		IF ABS(axis.NcToPlc.ActTorque) > ABS(TorqueLimit) THEN
			//fbDetectTime(IN := TRUE,PT := DetectionTorqueTime); 
			fbDetectTime.IN := TRUE;
			IF fbDetectTime.Q THEN
				jog.JogForward := FALSE;
				jog.JogBackwards := FALSE;
				nState := nState + 1;
			END_IF
		ELSIF NOT jogOut.Busy AND jogOut.Error THEN
			Error := jogOut.Error;
			ErrorID := jogOut.ErrorID;
			jog.JogForward := FALSE;
			jog.JogBackwards := FALSE;
			nState := 0;
		ELSIF jogOut.CommandAborted THEN
			jog.JogForward := FALSE;
			jog.JogBackwards := FALSE;
		ELSE
			fbDetectTime.IN := FALSE;
			//fbDetectTime(IN := FALSE,PT := DetectionTorqueTime);
		END_IF
		
	2: // Stop motor
		stop.Execute := TRUE;
		
		IF stopOut.Busy AND stopOut.Done THEN
			stop.Execute := FALSE;
			Busy := FALSE;
			Done := TRUE;
			nState := 0;
			
		ELSIF NOT stopOut.Busy AND stopOut.Error THEN
			Error := stopOut.Error;
			ErrorId := stopOut.ErrorID;
			stop.Execute := FALSE;
			nState := 0;
		END_IF
END_CASE

IF axis.Status.Error THEN
	nState := 0;
END_IF

ACTION actMove:
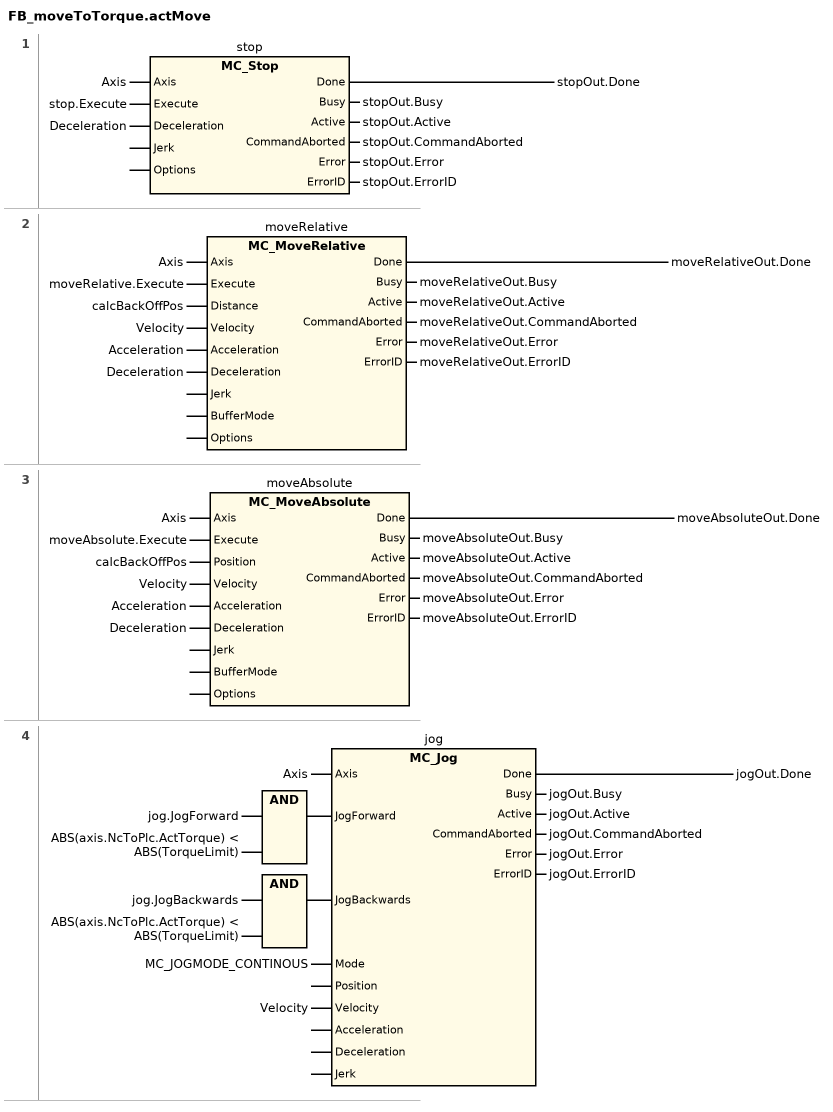
// NETWORK 1
stop(
    Axis := Axis,
    Execute := stop.Execute,
    Deceleration := Deceleration,
    Busy => stopOut.Busy,
    Active => stopOut.Active,
    CommandAborted => stopOut.CommandAborted,
    Error => stopOut.Error,
    ErrorID => stopOut.ErrorID); // MC_Stop
stopOut.Done := stop.Done;

// NETWORK 2
moveRelative(
    Axis := Axis,
    Execute := moveRelative.Execute,
    Distance := calcBackOffPos,
    Velocity := Velocity,
    Acceleration := Acceleration,
    Deceleration := Deceleration,
    Busy => moveRelativeOut.Busy,
    Active => moveRelativeOut.Active,
    CommandAborted => moveRelativeOut.CommandAborted,
    Error => moveRelativeOut.Error,
    ErrorID => moveRelativeOut.ErrorID); // MC_MoveRelative
moveRelativeOut.Done := moveRelative.Done;

// NETWORK 3
moveAbsolute(
    Axis := Axis,
    Execute := moveAbsolute.Execute,
    Position := calcBackOffPos,
    Velocity := Velocity,
    Acceleration := Acceleration,
    Deceleration := Deceleration,
    Busy => moveAbsoluteOut.Busy,
    Active => moveAbsoluteOut.Active,
    CommandAborted => moveAbsoluteOut.CommandAborted,
    Error => moveAbsoluteOut.Error,
    ErrorID => moveAbsoluteOut.ErrorID); // MC_MoveAbsolute
moveAbsoluteOut.Done := moveAbsolute.Done;

// NETWORK 4
jog(
    Axis := Axis,
    JogForward := jog.JogForward AND (ABS(axis.NcToPlc.ActTorque) < ABS(TorqueLimit)),
    JogBackwards := jog.JogBackwards AND (ABS(axis.NcToPlc.ActTorque) < ABS(TorqueLimit)),
    Mode := MC_JOGMODE_CONTINOUS,
    Velocity := Velocity,
    Busy => jogOut.Busy,
    Active => jogOut.Active,
    CommandAborted => jogOut.CommandAborted,
    Error => jogOut.Error,
    ErrorID => jogOut.ErrorID); // MC_Jog
jogOut.Done := jog.Done;
END_ACTION

END_FUNCTION_BLOCK

// ---- POUs/FUNCTIONS/FB_homeToTorque.TcPOU
FUNCTION_BLOCK FB_homeToTorque
VAR_IN_OUT
	Axis : AXIS_REF;					
END_VAR
VAR_INPUT
	Execute 		: BOOL;
	Direction 		: INT; // 0- PositiveDirection, 1- NegativeDirection
	Velocity 		: LREAL;
	Acceleration 	: LREAL;
	Deceleration 	: LREAL;
	SetPosition 	: LREAL;
	TimeLimit 		: TIME;
	TorqueLimit 	: LREAL;
	BackOffPos 		: LREAL;
END_VAR
VAR_OUTPUT
	Done 			: BOOL;
	Busy 			: BOOL;
	Active 			: BOOL;
	CommandAborted 	: BOOL;
	Error 			: BOOL;
	ErrorID 		: UDINT;
END_VAR
VAR
	nState 			: INT;
	fbExecute 		: R_TRIG;
	fbTimeout 		: TON;
	fbDetectTime 	: TON;
	
	readParameter 		: MC_ReadParameter;
	readParameterOut 	: ST_mcOutputs;
	
	writeParameter		: MC_WriteParameter;
	writeParameterOut 	: ST_mcOutputs;
	readValue 			: LREAL;
	
	parameter 	: MC_AxisParameter;	
	writeValue 	: LREAL;
	
	moveToTorque	: MC_TorqueControl;
	torqueOptions 	: ST_TorqueControlOptions;
	moveToTorqueOut : ST_mcOutputs;
	
	moveAbsolute	: MC_MoveAbsolute;
	moveAbsoluteOut : ST_mcOutputs;
	calcBackOffPos 	: LREAL;
	
	home	: MC_Home;
	homeOut : ST_mcOutputs;
	
	stop		: MC_Stop;
	stopOut 	: ST_mcOutputs;
	fPosition	: LREAL;

	jog		: MC_Jog;
	jogOut 	: ST_mcOutputs;
	
	moveRelative	: MC_MoveRelative;
	moveRelativeOut	: ST_mcOutputs;
END_VAR

fbExecute(CLK := Execute);
fbTimeout();
actHome();
actMode();
actMove();


CASE nState OF 
	0: //init
		IF NOT Execute THEN
		(* reset at falling edge of Execute *)
			Busy 					:= FALSE;
			Done					:= FALSE;
			CommandAborted 			:= FALSE;
			Error 					:= FALSE;
			ErrorID 				:= 0;
			fbTimeout.IN 			:= FALSE;
			readParameter.Enable 	:= FALSE;
			writeParameter.Execute	:= FALSE;
			stop.Execute		 	:= FALSE;
			home.Execute 			:= FALSE;
			moveAbsolute.Execute 	:= FALSE;
			jog.JogForward 			:= FALSE;
			jog.JogBackwards 		:= FALSE;
		END_IF
	
		IF fbExecute.Q THEN
			Busy := TRUE;
			nState := nState + 1;
		END_IF
		
	1:// Read soft limit switch to set back to when done
		CASE Direction OF 
			0: //mcPositiveDirection
		      	parameter := AxisMaxSoftPosLimit;
			1: //mcNegativeDirection
				parameter := AxisMinSoftPosLimit;
		END_CASE
		
		readParameter.Enable := TRUE;
		
		IF NOT readParameterOut.Busy AND readParameterOut.Done THEN
			readParameter.Enable := FALSE;
			nState := nState + 1;
		ELSIF NOT readParameterOut.Busy AND readParameterOut.Error THEN
			Error := readParameterOut.Error;
			ErrorId := readParameterOut.ErrorID;
			readParameter.Enable := FALSE;
			nState := 0;
		END_IF
		
	2: // Set soft limit switch to appropriate allowance
		CASE Direction OF
			0 : //mcPositiveDirection
				writeValue := 99999;
			1 : //mcNegativeDirection
				writeValue := -99999;
		END_CASE
		
		writeParameter.Execute := TRUE;
		
		IF NOT writeParameterOut.Busy AND writeParameterOut.Done THEN
			writeParameter.Execute := FALSE;
			nState := nState + 1;
		ELSIF NOT writeParameterOut.Busy AND writeParameterOut.Error THEN
			Error := writeParameterOut.Error;
			ErrorID := writeParameterOut.ErrorID;
			writeParameter.Execute := FALSE;
			nState := 0;
		END_IF
		
	3: //Execute MoveTowards Torque
		fbTimeout(IN:= TRUE, PT:= TimeLimit);
		
		CASE Direction OF
			0: //mcPositiveDirection 
				jog.JogForward := TRUE;
				jog.JogBackwards := FALSE;
			1: //mcNegativeDirection 
				jog.JogForward := FALSE;
				jog.JogBackwards := TRUE;
		END_CASE
			
		IF ABS(axis.NcToPlc.ActTorque) > ABS(TorqueLimit) THEN
			jog.JogForward := FALSE;
			jog.JogBackwards := FALSE;
			nState := nState + 1;
		ELSIF NOT jogOut.Busy AND jogOut.Error THEN
			Error := jogOut.Error;
			ErrorID := jogOut.ErrorID;
			jog.JogForward := FALSE;
			jog.JogBackwards := FALSE;
			nState := 0;
		END_IF
		
		// Timeout Error
		IF fbTimeout.Q THEN
			jog.JogForward := FALSE;
			jog.JogBackwards := FALSE;
			Error := TRUE;
			ErrorID := 1;
			nState := 0;
		END_IF
		
		CommandAborted := jogOut.CommandAborted;
	4://Stop motor 
		stop.Execute := TRUE;
		
		IF stopOut.Busy AND stopOut.Done THEN
			stop.Execute := FALSE;
			CASE Direction OF
				0: //mcPositiveDirection 
					calcBackOffPos := -BackOffPos;
				1: //mcNegativeDirection 
					calcBackOffPos := BackOffPos;
			END_CASE
			nState := nState + 1;
			
		ELSIF NOT stopOut.Busy AND stopOut.Error THEN
			Error := stopOut.Error;
			ErrorId := stopOut.ErrorID;
			stop.Execute := FALSE;
			nState := 0;
		END_IF
		
		CommandAborted := stopOut.CommandAborted;
	6: //Set homing state and counts
		IF axis.status.StandStill THEN
			home.Execute := TRUE;
		END_IF
		
		IF NOT homeOut.Busy AND homeOut.Done THEN
			home.Execute := FALSE;
			nState := nState + 1;
		ELSIF NOT homeOut.Busy AND homeOut.Error THEN
			Error := homeOut.Error;
			ErrorId := homeOut.ErrorID;
			home.Execute := FALSE;
			nState := 0;
		END_IF
		
		CommandAborted := homeOut.CommandAborted;
	5: //Move off home slightly
		IF axis.status.StandStill THEN
			moveRelative.Execute := TRUE;
		END_IF
		
		IF NOT moveRelativeOut.Busy AND moveRelativeOut.Done THEN
			moveRelative.Execute := FALSE;
			nState := nState + 1;
		ELSIF NOT moveRelativeOut.Busy AND moveRelativeOut.Error THEN
			Error := moveRelativeOut.Error;
			ErrorId := moveRelativeOut.ErrorID;
			moveRelative.Execute := FALSE;
			nState := 0;
		END_IF
		
		CommandAborted := moveRelativeOut.CommandAborted;
	7: // Write limit switch to original Value
		writeValue := SetPosition;
		writeParameter.Execute := TRUE;
		
		IF NOT writeParameterOut.Busy AND writeParameterOut.Done THEN
			writeParameter.Execute := FALSE;
			Busy := FALSE;
			Done := TRUE;
			nState := 0;
		ELSIF NOT writeParameterOut.Busy AND writeParameterOut.Error THEN
			Error := writeParameterOut.Error;
			ErrorID := writeParameterOut.ErrorID;
			writeParameter.Execute := FALSE;
			nState := 0;
		END_IF
END_CASE

IF axis.Status.Error THEN
	nState := 0;
END_IF

ACTION actHome:
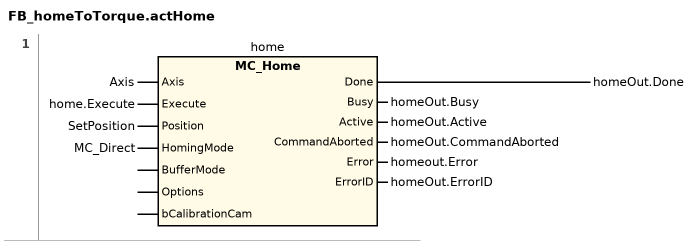
// NETWORK 1
home(
    Axis := Axis,
    Execute := home.Execute,
    Position := SetPosition,
    HomingMode := MC_Direct,
    Busy => homeOut.Busy,
    Active => homeOut.Active,
    CommandAborted => homeOut.CommandAborted,
    Error => homeout.Error,
    ErrorID => homeOut.ErrorID); // MC_Home
homeOut.Done := home.Done;
END_ACTION

ACTION actMode:
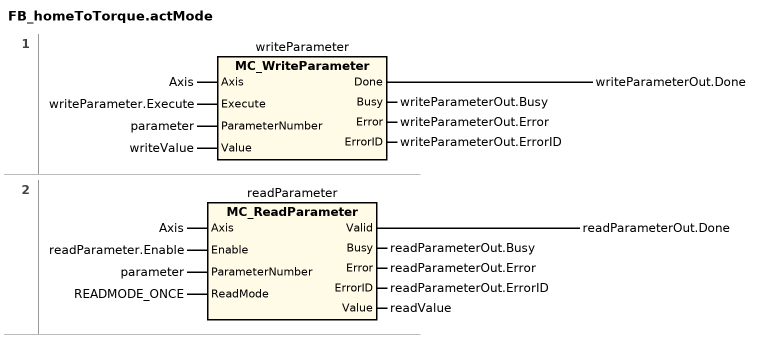
// NETWORK 1
writeParameter(
    Axis := Axis,
    Execute := writeParameter.Execute,
    ParameterNumber := parameter,
    Value := writeValue,
    Busy => writeParameterOut.Busy,
    Error => writeParameterOut.Error,
    ErrorID => writeParameterOut.ErrorID); // MC_WriteParameter
writeParameterOut.Done := writeParameter.Done;

// NETWORK 2
readParameter(
    Axis := Axis,
    Enable := readParameter.Enable,
    ParameterNumber := parameter,
    ReadMode := READMODE_ONCE,
    Busy => readParameterOut.Busy,
    Error => readParameterOut.Error,
    ErrorID => readParameterOut.ErrorID,
    Value => readValue); // MC_ReadParameter
readParameterOut.Done := readParameter.Valid;
END_ACTION

ACTION actMove:
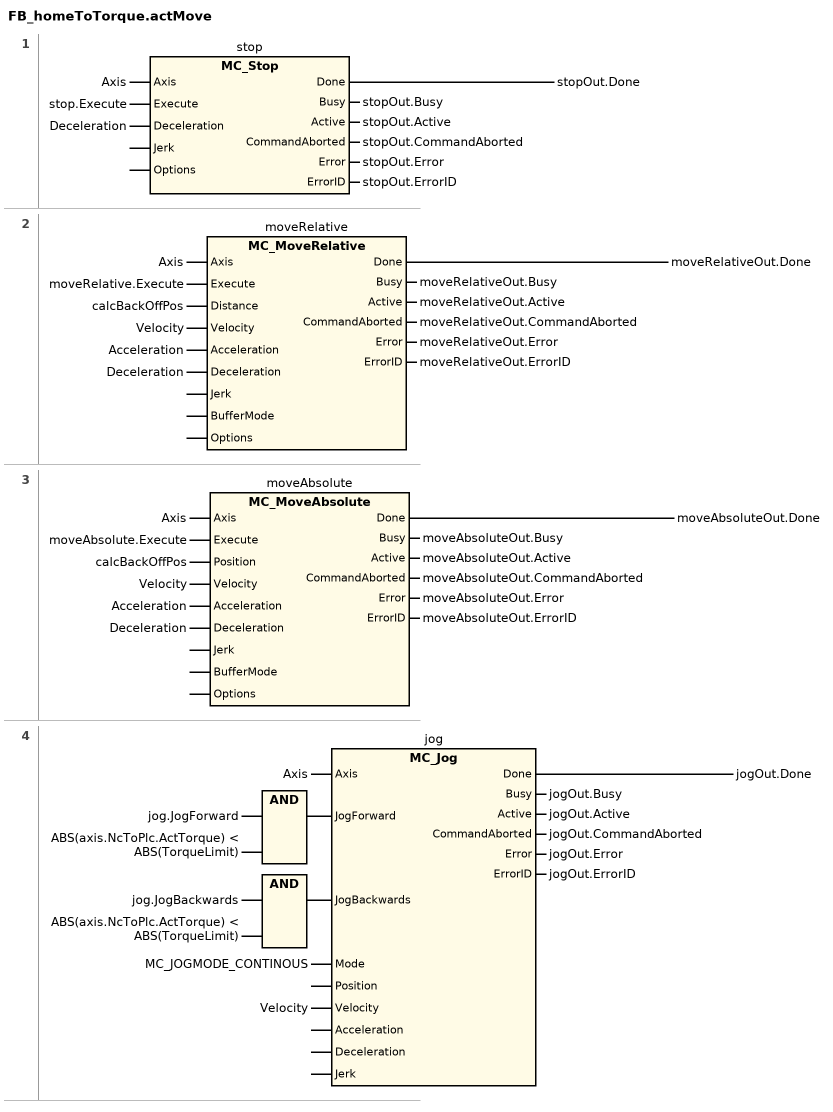
// NETWORK 1
stop(
    Axis := Axis,
    Execute := stop.Execute,
    Deceleration := Deceleration,
    Busy => stopOut.Busy,
    Active => stopOut.Active,
    CommandAborted => stopOut.CommandAborted,
    Error => stopOut.Error,
    ErrorID => stopOut.ErrorID); // MC_Stop
stopOut.Done := stop.Done;

// NETWORK 2
moveRelative(
    Axis := Axis,
    Execute := moveRelative.Execute,
    Distance := calcBackOffPos,
    Velocity := Velocity,
    Acceleration := Acceleration,
    Deceleration := Deceleration,
    Busy => moveRelativeOut.Busy,
    Active => moveRelativeOut.Active,
    CommandAborted => moveRelativeOut.CommandAborted,
    Error => moveRelativeOut.Error,
    ErrorID => moveRelativeOut.ErrorID); // MC_MoveRelative
moveRelativeOut.Done := moveRelative.Done;

// NETWORK 3
moveAbsolute(
    Axis := Axis,
    Execute := moveAbsolute.Execute,
    Position := calcBackOffPos,
    Velocity := Velocity,
    Acceleration := Acceleration,
    Deceleration := Deceleration,
    Busy => moveAbsoluteOut.Busy,
    Active => moveAbsoluteOut.Active,
    CommandAborted => moveAbsoluteOut.CommandAborted,
    Error => moveAbsoluteOut.Error,
    ErrorID => moveAbsoluteOut.ErrorID); // MC_MoveAbsolute
moveAbsoluteOut.Done := moveAbsolute.Done;

// NETWORK 4
jog(
    Axis := Axis,
    JogForward := jog.JogForward AND (ABS(axis.NcToPlc.ActTorque) < ABS(TorqueLimit)),
    JogBackwards := jog.JogBackwards AND (ABS(axis.NcToPlc.ActTorque) < ABS(TorqueLimit)),
    Mode := MC_JOGMODE_CONTINOUS,
    Velocity := Velocity,
    Busy => jogOut.Busy,
    Active => jogOut.Active,
    CommandAborted => jogOut.CommandAborted,
    Error => jogOut.Error,
    ErrorID => jogOut.ErrorID); // MC_Jog
jogOut.Done := jog.Done;
END_ACTION

END_FUNCTION_BLOCK

// ---- POUs/FUNCTIONS/FB_homeToSensorCustom.TcPOU
FUNCTION_BLOCK FB_homeToSensorCustom
VAR_IN_OUT
	Axis : AXIS_REF;					
END_VAR
VAR_INPUT
	Execute 		: BOOL;
	Direction 		: INT; // 0- PositiveDirection, 1- NegativeDirection
	Velocity 		: LREAL;
	Acceleration 	: LREAL;
	Deceleration 	: LREAL;
	SetPosition 	: LREAL;
	TimeLimit 		: TIME;
	TorqueLimit 	: LREAL;
	BackOffPos 		: LREAL;
	homeSensor		: BOOL;
END_VAR
VAR_OUTPUT
	Done 			: BOOL;
	Busy 			: BOOL;
	Active 			: BOOL;
	CommandAborted 	: BOOL;
	Error 			: BOOL;
	ErrorID 		: UDINT;
END_VAR
VAR
	nState 			: INT;
	fbExecute 		: R_TRIG;
	fbTimeout 		: TON;
	fbDetectTime 	: TON;
	
	readParameter 		: MC_ReadParameter;
	readParameterOut 	: ST_mcOutputs;
	
	writeParameter		: MC_WriteParameter;
	writeParameterOut 	: ST_mcOutputs;
	readValue 			: LREAL;
	
	parameter 	: MC_AxisParameter;	
	writeValue 	: LREAL;
	
	moveToTorque	: MC_TorqueControl;
	torqueOptions 	: ST_TorqueControlOptions;
	moveToTorqueOut : ST_mcOutputs;
	
	moveAbsolute	: MC_MoveAbsolute;
	moveAbsoluteOut : ST_mcOutputs;
	calcBackOffPos 	: LREAL;
	
	home	: MC_Home;
	homeOut : ST_mcOutputs;
	
	stop		: MC_Stop;
	stopOut 	: ST_mcOutputs;
	fPosition	: LREAL;

	jog		: MC_Jog;
	jogOut 	: ST_mcOutputs;
	
	moveRelative	: MC_MoveRelative;
	moveRelativeOut	: ST_mcOutputs;
END_VAR

// Copy of FB_homeToTorque but torque homing indicator is replaced with a homing sensor connected to the motor class. 
//Similiar to homeToSensor() method found in motor class. This function works better with motors that are not inverted. (ie motors that gain positive counts when moving away from their home position).
//homeToSensor() uses built in beckhoff homing function and works well when motor is invereted. I could not find a way to switch the direction of the homing back off after sensor was found so I created
//this custom function that accomplishes the same thing. 

fbExecute(CLK := Execute);
fbTimeout();
actHome();
actMode();
actMove();


CASE nState OF 
	0: //init
		IF NOT Execute THEN
		(* reset at falling edge of Execute *)
			Busy 					:= FALSE;
			Done					:= FALSE;
			CommandAborted 			:= FALSE;
			Error 					:= FALSE;
			ErrorID 				:= 0;
			fbTimeout.IN 			:= FALSE;
			readParameter.Enable 	:= FALSE;
			writeParameter.Execute	:= FALSE;
			stop.Execute		 	:= FALSE;
			home.Execute 			:= FALSE;
			moveAbsolute.Execute 	:= FALSE;
			jog.JogForward 			:= FALSE;
			jog.JogBackwards 		:= FALSE;
		END_IF
	
		IF fbExecute.Q THEN
			Busy := TRUE;
			nState := nState + 1;
		END_IF
		
	1:// Check homeSensor
		(*IF homeSensor THEN
			nState := 6;
		ELSE 
			nState := nState + 1;
		END_IF*)
		nState := nState + 1;
	2:// Read soft limit switch to set back to when done
		CASE Direction OF 
			0: //mcPositiveDirection
		      	parameter := AxisMaxSoftPosLimit;
			1: //mcNegativeDirection
				parameter := AxisMinSoftPosLimit;
		END_CASE
		
		readParameter.Enable := TRUE;
		
		IF NOT readParameterOut.Busy AND readParameterOut.Done THEN
			readParameter.Enable := FALSE;
			nState := nState + 1;
		ELSIF NOT readParameterOut.Busy AND readParameterOut.Error THEN
			Error := readParameterOut.Error;
			ErrorId := readParameterOut.ErrorID;
			readParameter.Enable := FALSE;
			nState := 0;
		END_IF
		
	3: // Set soft limit switch to appropriate allowance
		CASE Direction OF
			0 : //mcPositiveDirection
				writeValue := 99999;
			1 : //mcNegativeDirection
				writeValue := -99999;
		END_CASE
		
		writeParameter.Execute := TRUE;
		
		IF NOT writeParameterOut.Busy AND writeParameterOut.Done THEN
			writeParameter.Execute := FALSE;
			nState := nState + 1;
		ELSIF NOT writeParameterOut.Busy AND writeParameterOut.Error THEN
			Error := writeParameterOut.Error;
			ErrorID := writeParameterOut.ErrorID;
			writeParameter.Execute := FALSE;
			nState := 0;
		END_IF
		
	4: //Execute MoveTowards Sensor
		fbTimeout(IN:= TRUE, PT:= TimeLimit);
		
		CASE Direction OF
			0: //mcPositiveDirection 
				jog.JogForward := TRUE;
				jog.JogBackwards := FALSE;
			1: //mcNegativeDirection 
				jog.JogForward := FALSE;
				jog.JogBackwards := TRUE;
		END_CASE
			
		IF homeSensor THEN
			jog.JogForward := FALSE;
			jog.JogBackwards := FALSE;
			nState := nState + 1;
		ELSIF NOT jogOut.Busy AND jogOut.Error THEN
			Error := jogOut.Error;
			ErrorID := jogOut.ErrorID;
			jog.JogForward := FALSE;
			jog.JogBackwards := FALSE;
			nState := 0;
		END_IF
		
		// Timeout Error
		IF fbTimeout.Q THEN
			jog.JogForward := FALSE;
			jog.JogBackwards := FALSE;
			Error := TRUE;
			ErrorID := 1;
			nState := 0;
		END_IF
		
		CommandAborted := jogOut.CommandAborted;
		
	5://Stop motor 
		stop.Execute := TRUE;
		
		IF stopOut.Busy AND stopOut.Done THEN
			stop.Execute := FALSE;
			CASE Direction OF
				0: //mcPositiveDirection 
					calcBackOffPos := -BackOffPos;
				1: //mcNegativeDirection 
					calcBackOffPos := BackOffPos;
			END_CASE
			nState := nState + 1;
			
		ELSIF NOT stopOut.Busy AND stopOut.Error THEN
			Error := stopOut.Error;
			ErrorId := stopOut.ErrorID;
			stop.Execute := FALSE;
			nState := 0;
		END_IF
		
		CommandAborted := stopOut.CommandAborted;
		
	7: //Set homing state and counts
		IF axis.status.StandStill THEN
			home.Execute := TRUE;
		END_IF
		
		IF NOT homeOut.Busy AND homeOut.Done THEN
			home.Execute := FALSE;
			nState := nState + 1;
		ELSIF NOT homeOut.Busy AND homeOut.Error THEN
			Error := homeOut.Error;
			ErrorId := homeOut.ErrorID;
			home.Execute := FALSE;
			nState := 0;
		END_IF
		
		CommandAborted := homeOut.CommandAborted;
		
	6: //Move off home slightly
		IF axis.status.StandStill THEN
			moveRelative.Execute := TRUE;
		END_IF
		
		IF NOT moveRelativeOut.Busy AND moveRelativeOut.Done THEN
			moveRelative.Execute := FALSE;
			nState := nState + 1;
		ELSIF NOT moveRelativeOut.Busy AND moveRelativeOut.Error THEN
			Error := moveRelativeOut.Error;
			ErrorId := moveRelativeOut.ErrorID;
			moveRelative.Execute := FALSE;
			nState := 0;
		END_IF
		
		CommandAborted := moveRelativeOut.CommandAborted;
		
	8: // Write limit switch to original Value
		writeValue := SetPosition;
		writeParameter.Execute := TRUE;
		
		IF NOT writeParameterOut.Busy AND writeParameterOut.Done THEN
			writeParameter.Execute := FALSE;
			Busy := FALSE;
			Done := TRUE;
			nState := 0;
		ELSIF NOT writeParameterOut.Busy AND writeParameterOut.Error THEN
			Error := writeParameterOut.Error;
			ErrorID := writeParameterOut.ErrorID;
			writeParameter.Execute := FALSE;
			nState := 0;
		END_IF
END_CASE

IF axis.Status.Error THEN
	nState := 0;
END_IF

ACTION actHome:
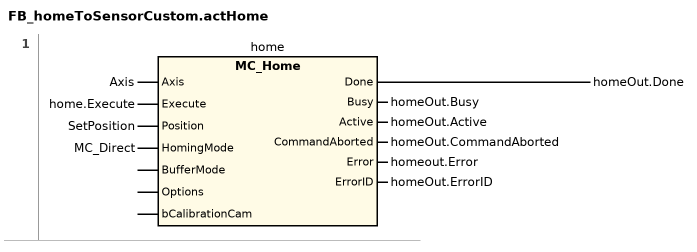
// NETWORK 1
home(
    Axis := Axis,
    Execute := home.Execute,
    Position := SetPosition,
    HomingMode := MC_Direct,
    Busy => homeOut.Busy,
    Active => homeOut.Active,
    CommandAborted => homeOut.CommandAborted,
    Error => homeout.Error,
    ErrorID => homeOut.ErrorID); // MC_Home
homeOut.Done := home.Done;
END_ACTION

ACTION actMode:
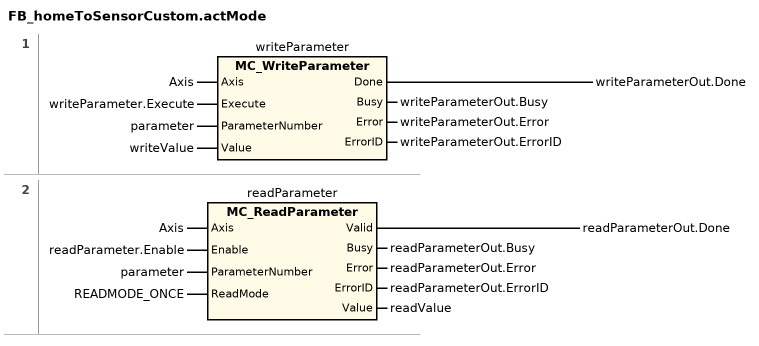
// NETWORK 1
writeParameter(
    Axis := Axis,
    Execute := writeParameter.Execute,
    ParameterNumber := parameter,
    Value := writeValue,
    Busy => writeParameterOut.Busy,
    Error => writeParameterOut.Error,
    ErrorID => writeParameterOut.ErrorID); // MC_WriteParameter
writeParameterOut.Done := writeParameter.Done;

// NETWORK 2
readParameter(
    Axis := Axis,
    Enable := readParameter.Enable,
    ParameterNumber := parameter,
    ReadMode := READMODE_ONCE,
    Busy => readParameterOut.Busy,
    Error => readParameterOut.Error,
    ErrorID => readParameterOut.ErrorID,
    Value => readValue); // MC_ReadParameter
readParameterOut.Done := readParameter.Valid;
END_ACTION

ACTION actMove:
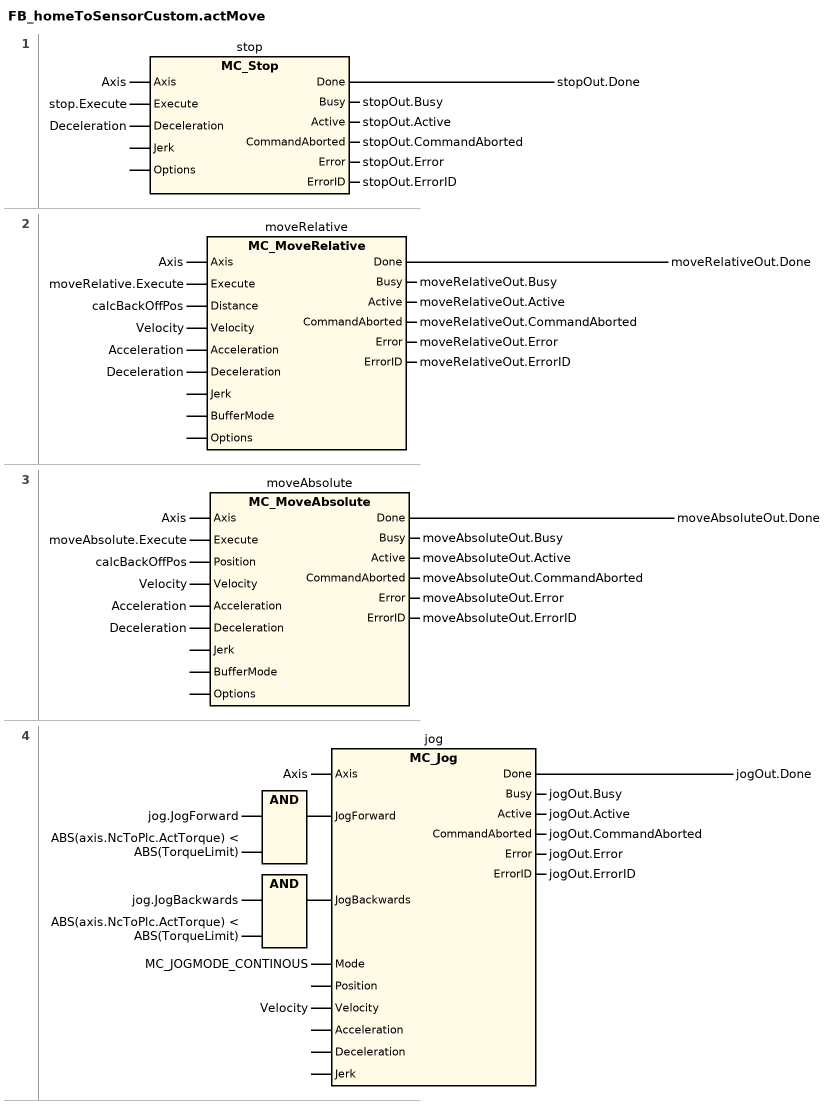
// NETWORK 1
stop(
    Axis := Axis,
    Execute := stop.Execute,
    Deceleration := Deceleration,
    Busy => stopOut.Busy,
    Active => stopOut.Active,
    CommandAborted => stopOut.CommandAborted,
    Error => stopOut.Error,
    ErrorID => stopOut.ErrorID); // MC_Stop
stopOut.Done := stop.Done;

// NETWORK 2
moveRelative(
    Axis := Axis,
    Execute := moveRelative.Execute,
    Distance := calcBackOffPos,
    Velocity := Velocity,
    Acceleration := Acceleration,
    Deceleration := Deceleration,
    Busy => moveRelativeOut.Busy,
    Active => moveRelativeOut.Active,
    CommandAborted => moveRelativeOut.CommandAborted,
    Error => moveRelativeOut.Error,
    ErrorID => moveRelativeOut.ErrorID); // MC_MoveRelative
moveRelativeOut.Done := moveRelative.Done;

// NETWORK 3
moveAbsolute(
    Axis := Axis,
    Execute := moveAbsolute.Execute,
    Position := calcBackOffPos,
    Velocity := Velocity,
    Acceleration := Acceleration,
    Deceleration := Deceleration,
    Busy => moveAbsoluteOut.Busy,
    Active => moveAbsoluteOut.Active,
    CommandAborted => moveAbsoluteOut.CommandAborted,
    Error => moveAbsoluteOut.Error,
    ErrorID => moveAbsoluteOut.ErrorID); // MC_MoveAbsolute
moveAbsoluteOut.Done := moveAbsolute.Done;

// NETWORK 4
jog(
    Axis := Axis,
    JogForward := jog.JogForward AND (ABS(axis.NcToPlc.ActTorque) < ABS(TorqueLimit)),
    JogBackwards := jog.JogBackwards AND (ABS(axis.NcToPlc.ActTorque) < ABS(TorqueLimit)),
    Mode := MC_JOGMODE_CONTINOUS,
    Velocity := Velocity,
    Busy => jogOut.Busy,
    Active => jogOut.Active,
    CommandAborted => jogOut.CommandAborted,
    Error => jogOut.Error,
    ErrorID => jogOut.ErrorID); // MC_Jog
jogOut.Done := jog.Done;
END_ACTION

END_FUNCTION_BLOCK

// ---- POUs/DEVICES/FB_ltBar.TcPOU
FUNCTION_BLOCK FB_ltBar
VAR
	bGreenLight 	AT %Q* : BOOL;
	bRedLight 		AT %Q* : BOOL;
	bYellowLight 	AT %Q* : BOOL;
END_VAR

METHOD greenOn : BOOL
VAR_INPUT
END_VAR
bGreenLight 	:= TRUE;
bRedLight 		:= FALSE;
bYellowLight 	:= FALSE;
END_METHOD

METHOD redOn : BOOL
VAR_INPUT
END_VAR
bGreenLight 	:= FALSE;
bRedLight 		:= TRUE;
bYellowLight 	:= FALSE;
END_METHOD

METHOD yellowOn : BOOL
VAR_INPUT
END_VAR
bGreenLight 	:= FALSE;
bRedLight 		:= FALSE;
bYellowLight 	:= TRUE;
END_METHOD

END_FUNCTION_BLOCK

// ---- POUs/DEVICES/FB_ltCurtains.TcPOU
FUNCTION_BLOCK FB_ltCurtains EXTENDS FB_pushBtnNC
VAR
	bLftCurtainFbError 		AT %I* : BOOL;
	bLftCurtainSigOk 		AT %I* : BOOL;
	bRhtCurtainFbError 		AT %I* : BOOL;
	bRhtCurtainSigOk 		AT %I* : BOOL;
	nLftCurtainFbState 		AT %I* : USINT; //States : 1 - Running, 2 - PreOp, 3 - Triggered, 6 - Reset 
	nRhtCurtainFbState 		AT %I* : USINT; //States : 1 - Running, 2 - PreOp, 3 - Triggered, 6 - Reset 
	

	bRhtCurtainEnable	AT %Q* : BOOL;
	bLftCurtainEnable	AT %Q* : BOOL;
	bResetLftCurtainFb 	AT %Q* : BOOL;
	bResetRhtCurtainFb 	AT %Q* : BOOL;
	bMuteCurtains 		AT %Q* : BOOL;
	
	bCurtainsMuted		AT %I* : BOOL;
	
END_VAR

PROPERTY curtainsMuted : BOOL
GET
curtainsMuted := bCurtainsMuted;
END_GET
END_PROPERTY

PROPERTY enableLftCurtain : BOOL
SET
bLftCurtainEnable := enableLftCurtain;
END_SET
END_PROPERTY

PROPERTY enableRhtCurtain : BOOL
SET
bRhtCurtainEnable := enableRhtCurtain;
END_SET
END_PROPERTY

METHOD mute : BOOL
VAR_INPUT
END_VAR
bMuteCurtains := TRUE;
mute := TRUE;
END_METHOD

METHOD reset : BOOL
VAR_INPUT
END_VAR
reset := FALSE;
bResetLftCurtainFb 	:= TRUE;
bResetRhtCurtainFb 	:= TRUE;

(*IF NOT GVL_machine.bLightCurtainsOk THEN
	bResetLftCurtainFb 	:= FALSE;
	bResetRhtCurtainFb 	:= FALSE;
	reset := TRUE;
END_IF*)
END_METHOD

PROPERTY resetLftCurtainFB : BOOL
SET
bResetLftCurtainFb := resetLftCurtainFB;
END_SET
END_PROPERTY

PROPERTY resetRhtCurtainFB : BOOL
SET
bResetRhtCurtainFb := resetRhtCurtainFB;
END_SET
END_PROPERTY

METHOD unmute : BOOL
VAR_INPUT
END_VAR
bMuteCurtains := FALSE;
unmute := TRUE;
END_METHOD

END_FUNCTION_BLOCK

// ---- POUs/DEVICES/FB_pushBtnNC.TcPOU
FUNCTION_BLOCK FB_pushBtnNC
VAR
	bBtn AT %I* : BOOL;
END_VAR

PROPERTY isPressed : BOOL
GET
IF NOT bBtn THEN 
	isPressed := TRUE;
ELSE 
	isPressed := FALSE;
END_IF
END_GET
END_PROPERTY

END_FUNCTION_BLOCK

// ---- POUs/DEVICES/FB_estop.TcPOU
FUNCTION_BLOCK FB_estop EXTENDS FB_pushBtnNC
VAR
	bResetEstopFb 		AT %Q* : BOOL;
	bEstopFbError 		AT %I* : BOOL;
	bEstopSigOk 		AT %I* : BOOL;
	nEstopFbState		AT %I* : USINT; //States : 1 - Running, 2 - PreOp, 3 - Triggered, 6 - Reset 
END_VAR

METHOD reset : BOOL
VAR_INPUT
END_VAR
reset := FALSE;
bResetEstopFb := TRUE;
IF NOT bEstopFbError THEN
	bResetEstopFb := FALSE;
	reset := TRUE;
END_IF
END_METHOD

PROPERTY resetEstopFB : BOOL
SET
bResetEstopFb := resetEstopFB;
END_SET
END_PROPERTY

END_FUNCTION_BLOCK

// ---- POUs/DEVICES/FB_table.TcPOU
FUNCTION_BLOCK FB_table
VAR
	tableDistSens 	: FB_distSensor2011;
	bTableGreenWire	AT %Q* : BOOL;				
	bTableBlackWire	AT %Q* : BOOL;	
	bTableBlueWire 	AT %Q* : BOOL;	
	bSafetySensor1 	AT %I* : BOOL;
	bSafetySensor2   AT %I* : BOOL;
	bLoadedSensor AT %I* : BOOL;
	
	fbSpaLoadedTime 	: TON;
	fbSpaUnloadedTime 	: TON;
	heightSensorOffset : REAL := 5.875;
	//heightSensorOffset : REAL := 1.25;
END_VAR

METHOD estop : BOOL
VAR_INPUT
END_VAR
btableBlackWire 	:= FALSE;
btableBlueWire 		:= FALSE;
btableGreenWire 	:= FALSE;
END_METHOD

METHOD moveDown : BOOL
VAR_INPUT
	distance: REAL;
END_VAR
bTableGreenWire := FALSE;
// IF safetySensor1 OR safetySensor2 THEN
//moveDown := 3 
//ELSE 
	IF tableHeight > distance THEN 
		bTableBlackWire := TRUE;
		bTableBlueWire := TRUE;
		moveDown := FALSE;
	ELSE 
		bTableBlackWire := FALSE;
		bTableBlueWire := FALSE;
		moveDown := TRUE;
	END_IF
//END_IF
END_METHOD

METHOD moveTo : BOOL
VAR_INPUT
	distance: REAL;
END_VAR
//IF safetySensor1 OR safetySensor2 THEN
//moveDown := 3 
//ELSE 
	//IF tableDistSens.height> distance + 1 THEN 
	IF tableHeight > distance + 0.5 THEN 
		bTableBlackWire := TRUE;
		bTableBlueWire := TRUE;
		bTableGreenWire := FALSE;
		
	ELSE 
		bTableBlackWire := FALSE;
		bTableBlueWire := FALSE;
		
	END_IF
	
	IF tableHeight < distance - 0.5 THEN 
		bTableBlackWire := FALSE;
		bTableBlueWire := FALSE;
		bTableGreenWire := TRUE;
		
	ELSE
		bTableGreenWire := FALSE;
		
	END_IF
	
	IF tableHeight < distance + 0.5 AND tableHeight > distance - 0.5 THEN 
		moveTo := TRUE;
	ELSE 
		moveTo := FALSE;
	END_IF
//END_IF
END_METHOD

METHOD moveUp : BOOL
VAR_INPUT
	distance : REAL;
END_VAR
bTableBlackWire := FALSE;
bTableBlueWire := FALSE;
// IF safetySensor1 OR safetySensor2 THEN
//moveDown := 3 
//ELSE 
	IF tableHeight < distance THEN 
		bTableGreenWire := TRUE;
		moveUp := FALSE;
	ELSE
		bTableGreenWire := FALSE;
		moveUp := TRUE;
	END_IF
//END_IF
END_METHOD

PROPERTY spaLoaded : BOOL
GET
spaLoaded := FALSE;
fbSpaLoadedTime(PT := T#1M);

IF bLoadedSensor THEN
	fbSpaLoadedTime.IN := TRUE;
ELSE 
	fbSpaLoadedTime.IN := FALSE;
END_IF

IF fbSpaLoadedTime.Q THEN
	spaLoaded := TRUE;
ELSE
	spaLoaded := FALSE;
END_IF
END_GET
END_PROPERTY

PROPERTY spaUnloaded : BOOL
GET
spaUnLoaded := FALSE;
fbSpaUnloadedTime(PT := T#2M);

IF NOT bLoadedSensor THEN
	fbSpaUnloadedTime.IN := TRUE;
ELSE 
	fbSpaUnloadedTime.IN := FALSE;
END_IF

IF fbSpaUnloadedTime.Q THEN
	spaUnLoaded := TRUE;
ELSE
	spaUnLoaded := FALSE;
END_IF
END_GET
END_PROPERTY

PROPERTY tableHeight : REAL
GET
tableHeight:= tableDistSens.height + heightSensorOffset;
END_GET
END_PROPERTY

METHOD tempMoveDown : BOOL
VAR_INPUT
END_VAR
//IF NOT safetySensor1 AND safetySensor2 THEN 
bTableGreenWire 	:= FALSE;
bTableBlackWire 	:= TRUE;
bTableBlueWire 	:= TRUE;
//ELSE
//nothing
//END_IF
END_METHOD

METHOD tempMoveUp : BOOL
VAR_INPUT
END_VAR
//IF NOT safetySensor1 AND safetySensor2 THEN 
bTableBlackWire := FALSE;
bTableBlueWire := FALSE;
bTableGreenWire := TRUE;
//ELSE
//nothing
//END_IF
END_METHOD

METHOD tempSteadyState : BOOL
VAR_INPUT
END_VAR
bTableBlackWire := FALSE;
bTableBlueWire := FALSE;
bTableGreenWire := FALSE;
END_METHOD

END_FUNCTION_BLOCK

// ---- POUs/DEVICES/FB_distSensor2011.TcPOU
FUNCTION_BLOCK FB_distSensor2011
VAR
	nSensor AT %I* 	: INT;
	fHeightVal 		: REAL;
	fSensorAvg		: REAL;
	nAvgSensorCount : INT;
	fPrevHeight		: REAL;
	fLowBound 		: REAL := 257; // mm's at 4 mA on sensor
	fHighBound		: REAL := 1226; // mm's at 20 mA on sensor
END_VAR

PROPERTY height : REAL //Distance in inches
GET
//height := (((INT_TO_REAL(sensor)/32767)*3000)+50)/25.4;
IF nAvgSensorCount <= 25 THEN
	nAvgSensorCount := nAvgSensorCount + 1;
	fSensorAvg := fSensorAvg + ((INT_TO_REAL(nSensor))/25);
	fHeightVal := fPrevHeight;
	height := fPrevHeight;
ELSE 
	height := (((fSensorAvg/43519)*fHighBound)+fLowBound)/25.4;
	fPrevHeight := height;
	fSensorAvg := 0;
	nAvgSensorCount := 0;
	fHeightVal := height;
END_IF
END_GET
END_PROPERTY

END_FUNCTION_BLOCK

// ---- POUs/DEVICES/FB_digitalOut.TcPOU
FUNCTION_BLOCK FB_digitalOut
VAR
	bOutput AT %Q* : BOOL;
END_VAR

METHOD turnOff : BOOL
VAR_INPUT
END_VAR
bOutput := FALSE;
END_METHOD

METHOD turnOn : BOOL
VAR_INPUT
END_VAR
bOutput := TRUE;
END_METHOD

END_FUNCTION_BLOCK

// ---- POUs/DEVICES/FB_pushBtnNO.TcPOU
FUNCTION_BLOCK FB_pushBtnNO
VAR
	bBtn AT %I* : BOOL;
END_VAR

PROPERTY isPressed : BOOL
GET
IF bBtn THEN 
	isPressed := TRUE;
ELSE 
	isPressed := FALSE;
END_IF
END_GET
END_PROPERTY

END_FUNCTION_BLOCK

// ---- POUs/FUNCTIONS/FB_MultiMotorController.TcPOU
FUNCTION_BLOCK FB_MultiMotorController
VAR_INPUT
	bExecute : BOOL; // Used to execute command. If error occurs excecute must go false and true again to execute command again. 
	aMotorRef :ARRAY[1..4] OF POINTER TO FB_teknicMotorEC; // Array of addresses of up to four motors to control. *Fill array in order of index **Must fill entire array. Unused spots - enter 0.
	eMethod : E_teknicMotorMethods; // Method to call for control of specified motors
END_VAR
VAR_OUTPUT
	aDone 			: ARRAY[1..4] OF BOOL;
	aBusy			: ARRAY[1..4] OF BOOL;
	aError 			: ARRAY[1..4] OF BOOL;
	aErrorID 		: ARRAY[1..4] OF UDINT;
	sControllerMsg 	: STRING; // String used to display messages from the controller FB.
END_VAR
VAR
	fbExecute 		: R_TRIG;
	bDone: INT;
	i : INT;
END_VAR

(* Example call- FB_multiMotorController(bExecute := TRUE, aMotorRef := [ADR(FB_teknicMotor1),ADR(FB_teknicMotor2),0,0],sMethod := moveToJog); *)
fbExecute(CLK := bExecute);
IF NOT bExecute THEN
(* reset at falling edge of Execute *)
	aDone[1.4]				:= FALSE;
	aError[1.4] 			:= FALSE;
	aErrorID[1.4] 			:= 0;
END_IF
IF bExecute THEN		
	CASE eMethod OF 
		brakeOff://
			FOR i := 1 TO 4 BY 1 DO
				IF aMotorRef[i] <> 0 THEN
					IF aMotorRef[i]^.brakeOff() THEN
						aDone[i] := TRUE;
					END_IF
				END_IF
			END_FOR
			
		brakeOn://
			FOR i := 1 TO 4 BY 1 DO
				IF aMotorRef[i] <> 0 THEN
					IF aMotorRef[i]^.brakeOn() THEN
						aDone[i] := TRUE;
					END_IF
				END_IF
			END_FOR
		checkOutputs://
		coupleToAxis://
		decoupleAxis://
		disable://
			FOR i := 1 TO 4 BY 1 DO
				IF aMotorRef[i] <> 0 THEN
					CASE aMotorRef[i]^.disable() OF
						1:// Done
							aDone[i] := TRUE;
						13:// Error
							aError[i] := TRUE;	
					END_CASE
				END_IF
			END_FOR
		enable://
			FOR i := 1 TO 4 BY 1 DO
				IF aMotorRef[i] <> 0 THEN
					CASE aMotorRef[i]^.enable() OF
						1:// Done
							aDone[i] := TRUE;
						13:// Error
							aError[i] := TRUE;	
					END_CASE
				END_IF
			END_FOR
		estop://
		homeToSensor://
			FOR i := 1 TO 4 BY 1 DO
				IF aMotorRef[i] <> 0 THEN
					CASE aMotorRef[i]^.homeToSensor(0) OF
						1:// Done
							aDone[i] := TRUE;
						13:// Error
							aError[i] := TRUE;	
					END_CASE
				END_IF
			END_FOR
		homeToTorque://
			FOR i := 1 TO 4 BY 1 DO
				IF aMotorRef[i] <> 0 THEN
					CASE aMotorRef[i]^.homeToTorque() OF
						1:// Done
							aDone[i] := TRUE;
						3://Busy
							aBusy[i] := TRUE;
						13:// Error
							aError[i] := TRUE;	
					END_CASE
				END_IF
			END_FOR
		motorInit://
		moveTo://
		moveToJog://
		moveToSensor://
		moveToTorque://
		readMotorParameter://
			//sControllerMsg := LREAL_TO_STRING(aMotorRef[1]^.readValue);
		removeStop://
		motorReset://
		resetMotorCommands://
		setError://
		stop://
		writeMotorParameter://
	END_CASE
END_IF

END_FUNCTION_BLOCK

// ---- GlobalTextList.TcGTLO
TEXTLIST GlobalTextList
  150 = '%2.2f in.'
  1334 = '%2.2f percent'
  667 = '%2.3f in.'
  1379 = '%2.3f percent'
  330 = '%s'
  441 = 'A5L'
  558 = 'A6'
  483 = 'A7'
  986 = 'A8'
  298 = 'A9L'
  781 = 'Action is complete'
  1160 = 'ACTIVE'
  228 = 'Admin'
  94 = 'AUTO'
  924 = 'AUTOMATED A Series Flipper'
  62 = 'AUTOMATED A Series Flipper 2'
  33 = 'AWAY FROM \nHOME'
  979 = 'BACK'
  972 = 'BUSY'
  655 = 'BYPASS SAFETY'
  571 = 'CENTERING TORQUE'
  52 = 'CLAMP ON TORQUE'
  952 = 'CLAMP OPEN DIST'
  239 = 'CLAMPING'
  566 = 'CLEAR SAFETY'
  1017 = 'Click to Enable Motor Control'
  762 = 'Click to Enable Specified Motor Control'
  47 = 'Click to set position used for certain actions'
  260 = 'Click to set torque used for certain actions'
  659 = 'COLUMN'
  147 = 'COLUMN 0'
  332 = 'COLUMN 1'
  149 = 'COLUMN 2'
  796 = 'COLUMN 3'
  925 = 'COLUMN0'
  396 = 'COLUMN1'
  863 = 'COLUMNS'
  406 = 'CONFIRM'
  117 = 'CONTINUE'
  2 = 'CONTINUE\nPROGRAM'
  484 = 'CONTROL LOOP CLOSED'
  215 = 'CONTROLS'
  1037 = 'CONVEYOR HEIGHT IN'
  805 = 'COUPLED'
  127 = 'Current Height \n%5.2f'
  884 = 'Current Motor Position (measured in counts)'
  365 = 'Current Motor Position (mm)'
  76 = 'Current Motor Torque (measured in %)'
  91 = 'Current Rotation \n%5.2f'
  144 = 'Current Row : %2.0d'
  721 = 'Current speeds of motor (deg/s or mm/s)'
  980 = 'Current User: %s'
  258 = 'DISABLED'
  293 = 'DONE'
  183 = 'DRIVE DEVICE ERROR'
  644 = 'Drop down for desired \naction on motor'
  871 = 'Drop down for desired action on motor'
  1034 = 'EFLEX'
  853 = 'ENCODER : %f3.2'
  220 = 'ERROR'
  460 = 'ERROR '
  722 = 'ERROR DATA'
  210 = 'ERROR ID: '
  756 = 'ERROR ID: %3.2f'
  189 = 'ERROR ID: %5d'
  819 = 'ERROR ID: %f3.2'
  326 = 'Error is present in the current action'
  359 = 'ERROR MESSAGE'
  1027 = 'ERROR STOP'
  764 = 'ERRORS'
  348 = 'EXECUTE'
  357 = 'Function Block'
  791 = 'Hello '
  733 = 'HELP'
  7 = 'HLEP'
  636 = 'HOME'
  236 = 'HOMED'
  358 = 'ID'
  193 = 'INPUT'
  804 = 'Integer representation of error present '
  1061 = 'INVERTED'
  873 = 'Inverted = Negative Counts are away from home, Positive are towards home.'
  136 = 'KEEP AREA CLEAR'
  313 = 'Label'
  797 = 'LeFT CLAMP'
  911 = 'LEFT CLAMP'
  137 = 'LeFT ROTATION'
  583 = 'LEFT ROTATION'
  684 = 'LEFT ROTATION HOME SET POS'
  274 = 'LEFT WIDTH'
  363 = 'LFT CLAMP'
  222 = 'LFT CLAMPING'
  589 = 'LFT ROTATION'
  139 = 'LFT WIDTH'
  823 = 'LOGIN'
  288 = 'LOGOUT'
  119 = 'MACHINE SETTINGS'
  56 = 'MAIN'
  148 = 'MANTENER EL AREA DESPEJADA'
  53 = 'MANUAL'
  1074 = 'MANUAL\n (FULL CONTROL)'
  969 = 'MAP'
  1035 = 'MODE'
  1179 = 'MOTION COMMANDS LOCKED'
  356 = 'MOTOR'
  1159 = 'MOTOR\n (FULL CONTROL)'
  259 = 'MOTOR 1'
  55 = 'Motor is currently executing an action'
  645 = 'MOTORS STARTUP\nFAILED'
  349 = 'MOTORS STARTUP\nPlease wait...'
  166 = 'None'
  1483 = 'OPERATIONAL'
  1573 = 'Operator'
  225 = 'OPERTATIONAL'
  926 = 'OUTPUT'
  165 = 'PARAMETERS'
  631 = 'POSITION : %3.2f'
  975 = 'POSITION : %f3.2'
  677 = 'Position Input'
  738 = 'Previous Program Running. \n\nCONTINUE PROGRAM? '
  195 = 'PROTECTED MODE'
  669 = 'READ'
  30 = 'Read Value: %3.2f '
  342 = 'RESET'
  218 = 'RESET MACHINE'
  278 = 'RESET SAFETY'
  297 = 'RESTART\nPROGRAM'
  54 = 'RIGHT CLAMP'
  360 = 'RIGHT ROTATION'
  639 = 'RIGHT ROTATION HOME SET POS'
  20 = 'RIGHT WIDTH'
  427 = 'ROTATION'
  629 = 'SAFETY'
  932 = 'SAFETY BYPASSED'
  2143 = 'SAVE'
  1224 = 'Service'
  874 = 'Set Position'
  226 = 'Set Position used for certain actions'
  567 = 'Set Position: %3.2f'
  74 = 'Set Position: %3.2f '
  309 = 'Set Position: %3.2f in'
  1120 = 'Set Position: %3.2f in.'
  169 = 'Set Position: %f3.2'
  736 = 'Set Torque'
  240 = 'Set Torque used for certain actions'
  1146 = 'Set Torque: %3.2f'
  123 = 'Set Torque: %3.2f percent'
  878 = 'Set Torque: %f3.2'
  400 = 'SETTINGS'
  1296 = 'SOFT LIMIT MAX EXCEEDED'
  632 = 'SOFT LIMIT MIN EXCEEDED'
  1070 = 'SOLT LIMIT MIN EXCEEDED'
  542 = 'Spa Model: %s'
  485 = 'SPEED : %3.2f'
  717 = 'SPEED : %f3.2'
  317 = 'START'
  549 = 'STATUS'
  253 = 'STOP'
  42 = 'Supervisor'
  83 = 'TABLE'
  693 = 'TABLE CLAMPING HEIGHT'
  108 = 'TABLE DOWN HEIGHT'
  77 = 'Table Height : \n%5.2f'
  1466 = 'Team Lead'
  355 = 'TIME'
  917 = 'Toggle button to \nexecute selected action'
  235 = 'Toggle button to \nexecute/stop selected action'
  1092 = 'Toggle command to \nexecute selected action'
  876 = 'Toggle command to execute selected action'
  1213 = 'TORQUE : %3.2f'
  686 = 'TORQUE : %f3.2'
  1020 = 'TOWARDS\nHOME'
  430 = 'Variable Index: %3.0d'
  809 = 'Variable Index: %3f '
  810 = 'Variable Index: %3f.0d'
  385 = 'WARNING: Safety is not active!\nDo you wish to continue? '
  158 = 'WIDTH'
  1141 = 'WRITE'
  1195 = 'Write Value: %3.2f '
END_TEXTLIST

// ---- POUs/LISTS/actionSelectList.TcTLO
TEXTLIST actionSelectList
  0 = 'BRAKE OFF'
  1 = 'BRAKE ON'
  2 = 'DISABLE'
  3 = 'ENABLE'
  4 = 'HOME TO SENSOR'
  5 = 'HOME TO TORQUE'
  6 = 'MOVE TO POSITION'
  7 = 'JOG'
  8 = 'MOVE TO TORQUE'
  9 = 'RESET'
   = ''
END_TEXTLIST

// ---- VISUs/VISUs/Auto Screens/baseInSkiOutScreen.TcVIS
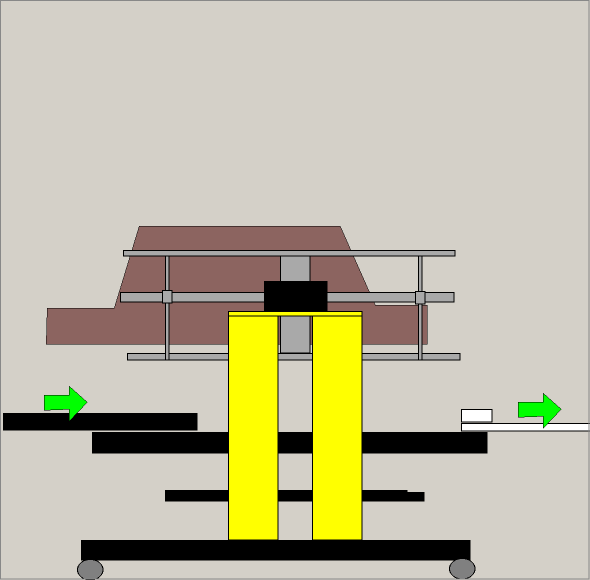
VISUALIZATION baseInSkiOutScreen  // 590x580
    Rectangle (461,423 130x8)
    Polygon (46,344) (47,308) (114,308) (139,226) (340,226) (375,305) (427,305) (427,343) (427,344)
    Rectangle (246,289 98x30), angle 90
    Rectangle (127,353 333x7)
    Rectangle (165,490 242x11), angle 25
    Rectangle (181,492 243x9), angle 336
    Rectangle (92,432 395x21)
    Rectangle (81,540 389x20)
    Rectangle (228,315 50x225)
    Rectangle (312,315 50x225)
    Ellipse (449,558 26x21)
    Ellipse (77,559 26x21)
    Rectangle (228,311 134x5)
    Rectangle (418,255 4x105)
    Rectangle (165,255 4x105)
    Rectangle (123,250 332x6)
    Rectangle (120,292 334x10)
    Rectangle (461,409 31x13)
    Rectangle (415,291 10x13)
    Rectangle (162,290 10x13)
    Rectangle (3,413 194x17)
    Polygon (44,405) (44,410) (69,409) (69,421) (87,402) (69,386) (69,395) (44,395)
    Polygon (518,412) (518,417) (543,416) (543,428) (561,409) (543,393) (543,402) (518,402)
    Rectangle (264,281 63x30)
END_VISUALIZATION

// ---- VISUs/VISUs/Auto Screens/continueAutoScreen.TcVIS
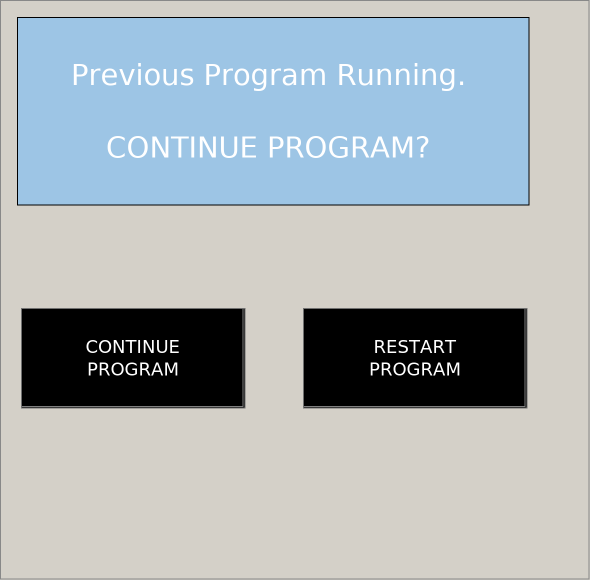
VISUALIZATION continueAutoScreen  // 590x580
    Textfield (17,17 512x188), "Previous Program Running. CONTINUE PROGRAM?"
    Button (21,308 224x100), "CONTINUE PROGRAM"
        toggle auto.bContinueProgBtn
    Button (303,308 224x100), "RESTART PROGRAM"
        toggle auto.bRestartProgBtn
END_VISUALIZATION

// ---- VISUs/VISUs/Auto Screens/eflexScreen.TcVIS
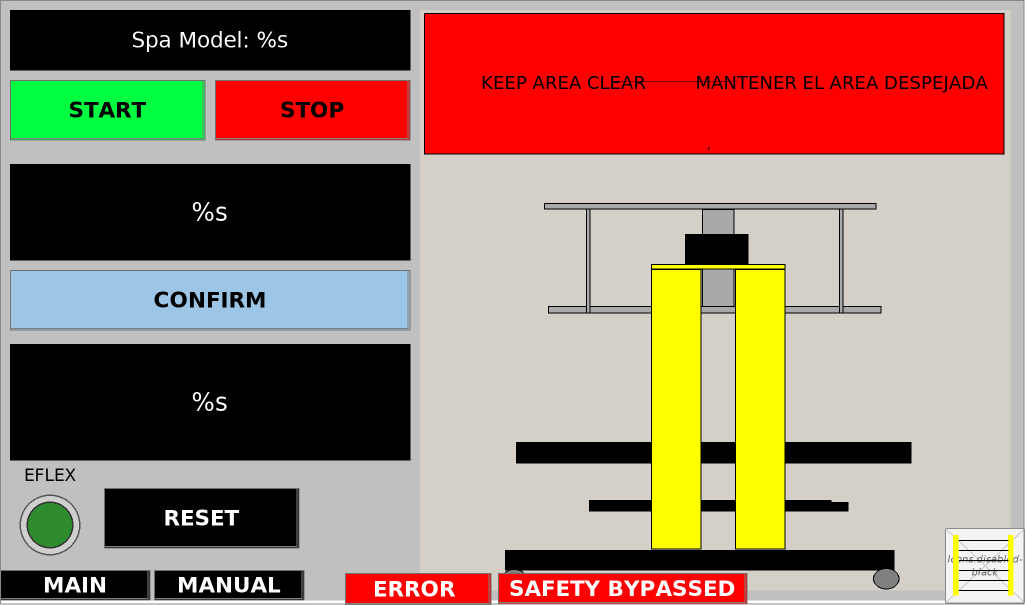
VISUALIZATION eflexScreen  // 1025x605
    Rectangle (0,0 1024x600)
    Button (0,570 150x30), "MAIN"
        OnMouseDown: change screen: mainScreen
        OnMouseDown: execute { GVL_machine.nPageIndex := 0; }
    Button (154,570 150x30), "MANUAL"
        OnMouseDown: change screen: manualScreen
        OnMouseDown: execute { GVL_machine.nPageIndex := 5; }
    RoundedRectangle (10,10 400x60), "Spa Model: %s", text variable: GVL_eflex.sSpaModel
    Button (10,80 195x60), "START", invisible if: auto.bHideStartBtn
        toggle auto.bStartBtn
    Button (215,80 195x60), "STOP", invisible if: auto.bHideStopBtn
        toggle auto.bStopBtn
    Frame (420,10 590x580), frame switch variable: auto.nFrameDisp
        shows machineHomingScreen()
        shows baseInSkiOutScreen()
        shows loadSpaScreen()
        shows studsInScreen()
        shows unloadSpaScreen()
        shows manualScreen()
        shows safetyResetScreen()
        shows tempEflexScreen()
        shows continueAutoScreen()
    Textfield (10,164 400x96), "%s", text variable: auto.sPromptDisp
    Button (10,270 400x60), "CONFIRM", invisible if: auto.bHideConfirmBtn
        tap auto.bConfirmBtn
    RoundedRectangle (0,460 100x30), "EFLEX"
    Lamp1 (15,490 70x70), variable: eflex.fbMqttClient.bConnected, style: Lamp-Lamp1-Green
    Button (104,488 195x60), "RESET"
        toggle auto.bResetBtn
    Button (498,573 249x31), "SAFETY BYPASSED", invisible if: NOT GVL_machine.bSafetyBypass
        OnMouseDown: change screen: safetyDisableWarning
    Button (345,573 146x32), "ERROR", invisible if: NOT GVL_machine.bDispErrorIcon
        OnMouseDown: change screen: errorScreen
    Image (945,528 80x75), invisible if: MAIN.bHideLtCurtainDisable, image: Icons.disabled-black
    Group (953,535 60x60), invisible if: GVL_machine.bSafetyBypass
        toggle GVL_machine.bMuteSafety
        Rectangle (0,0 5x60)
        Rectangle (55,0 5x60)
        Line (6,5) (55,5)
        Line (6,15) (55,15)
        Line (6,25) (55,25)
        Line (6,35) (55,35)
        Line (6,45) (55,45)
        Line (6,55) (55,55)
    Textfield (10,344 400x116), "%s", text variable: auto.sCheckDisp, invisible if: auto.bHideCheckDisp
END_VISUALIZATION

// ---- VISUs/VISUs/Auto Screens/loadSpaScreen.TcVIS
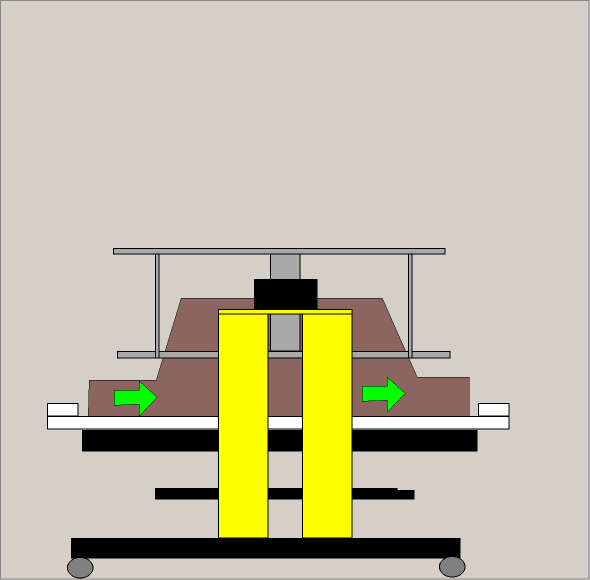
VISUALIZATION loadSpaScreen  // 590x580
    Rectangle (47,416 462x13)
    Polygon (88,416) (89,380) (156,380) (181,298) (382,298) (417,377) (469,377) (469,415) (469,416)
    Rectangle (236,287 98x30), angle 90
    Rectangle (117,351 333x7)
    Rectangle (155,488 242x11), angle 25
    Rectangle (171,490 243x9), angle 336
    Rectangle (82,430 395x21)
    Rectangle (71,538 389x20)
    Rectangle (218,313 50x225)
    Rectangle (302,313 50x225)
    Ellipse (439,556 26x21)
    Ellipse (67,557 26x21)
    Rectangle (218,309 134x5)
    Rectangle (254,279 63x30)
    Rectangle (408,253 4x105)
    Rectangle (155,253 4x105)
    Rectangle (113,248 332x6)
    Polygon (114,400) (114,405) (139,404) (139,416) (157,397) (139,381) (139,390) (114,390)
    Polygon (362,396) (362,401) (387,400) (387,412) (405,393) (387,377) (387,386) (362,386)
    Rectangle (478,403 31x13)
    Rectangle (47,403 31x13)
END_VISUALIZATION

// ---- VISUs/VISUs/Auto Screens/machineHomingScreen.TcVIS
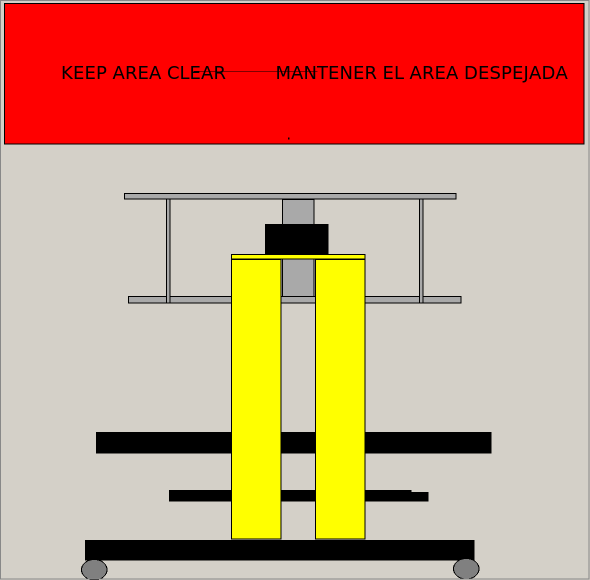
VISUALIZATION machineHomingScreen  // 590x580
    Rectangle (4,3 580x141)
    Rectangle (249,232 98x32), angle 90
    Rectangle (128,296 333x7)
    Rectangle (169,490 242x11), angle 25
    Rectangle (185,492 243x9), angle 336
    Rectangle (96,432 395x21)
    Rectangle (85,540 389x20)
    Rectangle (231,259 50x280)
    Rectangle (315,259 50x280)
    Ellipse (453,558 26x21)
    Ellipse (81,559 26x21)
    Rectangle (231,254 134x5)
    Rectangle (265,224 63x30)
    Rectangle (419,198 4x105)
    Rectangle (166,198 4x105)
    Rectangle (124,193 332x6)
    Label (18,48 251x50), "KEEP AREA CLEAR"
    Label (250,48 344x50), "MANTENER EL AREA DESPEJADA"
    Rectangle (288,138 1x0)
    Rectangle (194,71 123x0), angle 299
END_VISUALIZATION

// ---- VISUs/VISUs/Auto Screens/studsInScreen.TcVIS
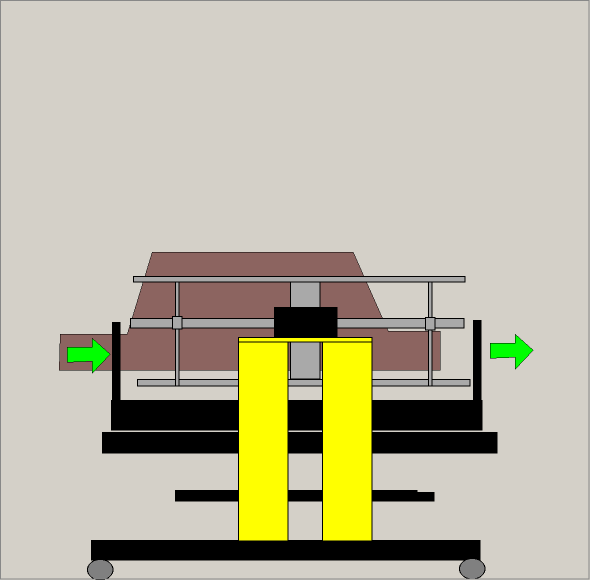
VISUALIZATION studsInScreen  // 590x580
    Polygon (59,370) (60,334) (127,334) (152,252) (353,252) (388,331) (440,331) (440,369) (440,370)
    Rectangle (111,400 371x30)
    Rectangle (256,315 98x30), angle 90
    Rectangle (137,379 333x7)
    Rectangle (175,490 242x11), angle 25
    Rectangle (191,492 243x9), angle 336
    Rectangle (102,432 395x21)
    Rectangle (91,540 389x20)
    Rectangle (238,341 50x200)
    Rectangle (322,341 50x200)
    Ellipse (459,558 26x21)
    Ellipse (87,559 26x21)
    Rectangle (238,337 134x5)
    Rectangle (428,281 4x105)
    Rectangle (175,281 4x105)
    Rectangle (133,276 332x6)
    Rectangle (130,318 334x10)
    Rectangle (425,317 10x13)
    Rectangle (172,316 10x13)
    Rectangle (274,307 63x30)
    Rectangle (473,320 8x101)
    Rectangle (112,322 8x101)
    Polygon (67,357) (67,362) (92,361) (92,373) (110,354) (92,338) (92,347) (67,347)
    Polygon (490,353) (490,358) (515,357) (515,369) (533,350) (515,334) (515,343) (490,343)
END_VISUALIZATION

// ---- VISUs/VISUs/Auto Screens/tempEflexScreen.TcVIS
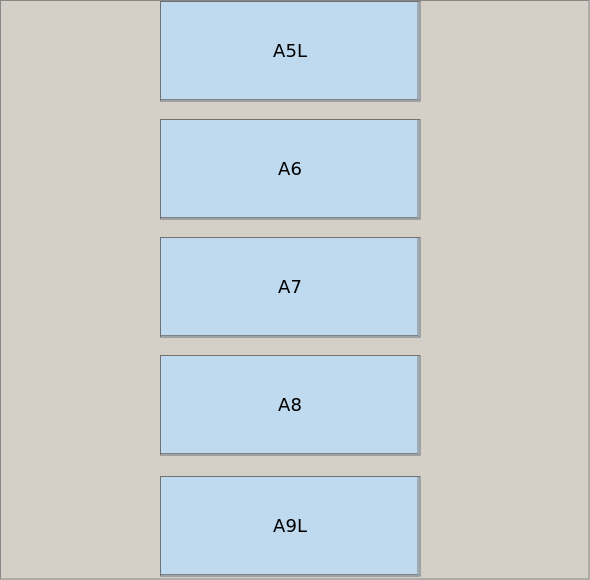
VISUALIZATION tempEflexScreen  // 590x580
    Button (160,1 260x100), "A5L"
        OnMouseDown: execute { tempEflex.nEflexState := 1; }
    Button (160,119 260x100), "A6"
        OnMouseDown: execute { tempEflex.nEflexState := 2; }
    Button (160,237 260x100), "A7"
        OnMouseDown: execute { tempEflex.nEflexState := 3; }
    Button (160,476 260x100), "A9L"
        OnMouseDown: execute { tempEflex.nEflexState := 5; }
    Button (160,355 260x100), "A8"
        OnMouseDown: execute { tempEflex.nEflexState := 4; }
END_VISUALIZATION

// ---- VISUs/VISUs/Auto Screens/unloadSpaScreen.TcVIS
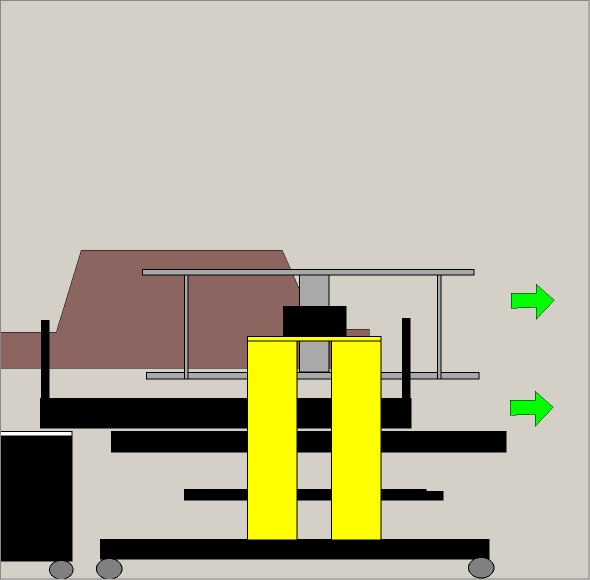
VISUALIZATION unloadSpaScreen  // 590x580
    Polygon (-12,368) (-11,332) (56,332) (81,250) (282,250) (317,329) (369,329) (369,367) (369,368)
    Rectangle (40,398 371x30)
    Rectangle (265,308 98x30), angle 90
    Rectangle (146,372 333x7)
    Rectangle (184,489 242x11), angle 25
    Rectangle (200,491 243x9), angle 336
    Rectangle (111,431 395x21)
    Rectangle (100,539 389x20)
    Rectangle (247,340 50x200)
    Rectangle (331,340 50x200)
    Ellipse (468,557 26x21)
    Ellipse (96,558 26x21)
    Rectangle (247,336 134x5)
    Rectangle (437,274 4x105)
    Rectangle (184,274 4x105)
    Rectangle (142,269 332x6)
    Rectangle (283,306 63x30)
    Rectangle (402,318 8x101)
    Rectangle (41,320 8x101)
    Polygon (511,303) (511,308) (536,307) (536,319) (554,300) (536,284) (536,293) (511,293)
    Polygon (510,410) (510,415) (535,414) (535,426) (553,407) (535,391) (535,400) (510,400)
    Rectangle (0,431 72x5)
    Rectangle (0,436 72x125)
    Ellipse (49,560 24x19)
END_VISUALIZATION

// ---- VISUs/VISUs/multiControlScreens/parametersScreen.TcVIS
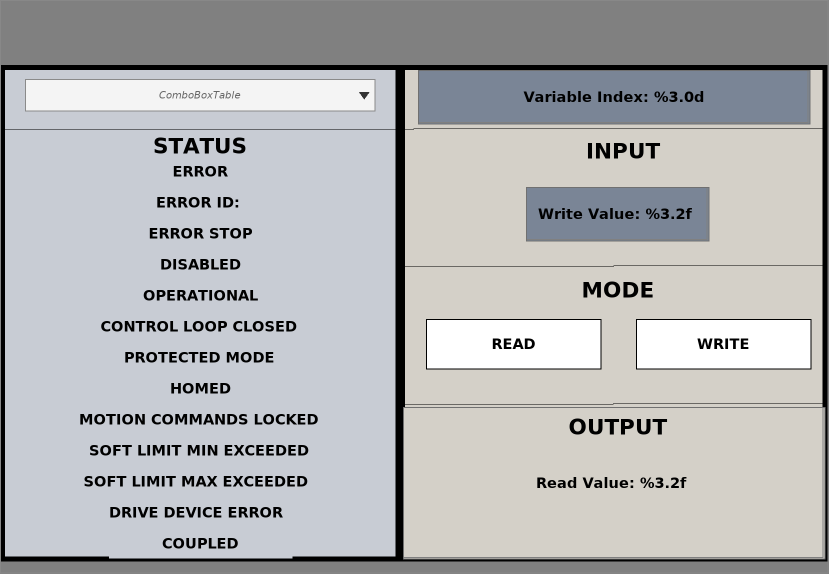
VISUALIZATION parametersScreen  // 829x574
    Rectangle (400,65 427x496)
    Button (403,407 422x152), "Read Value: %3.2f", text variable: multiControl.fValueOut
    Rectangle (0,65 400x496)
    Rectangle (109,281 183x29), "OPERATIONAL", colour toggle: multiControl.aStatusVar[4]
    Rectangle (109,374 183x29), "HOMED", colour toggle: multiControl.aStatusVar[7]
    Rectangle (74,312 250x29), "CONTROL LOOP CLOSED", colour toggle: multiControl.aStatusVar[5]
    Button (526,187 183x54), "Write Value: %3.2f", text variable: multiControl.fValueIn
        OnMouseClick: write the text variable via VisuDialogs.Numpad
    Line (0,129) (827,128)
    Line (402,266) (825,265)
    Line (401,404) (825,403)
    RoundedRectangle (426,319 175x50), "READ", colour toggle: multiControl.bReadParam
        toggle multiControl.bReadParam
    RoundedRectangle (636,319 175x50), "WRITE", colour toggle: multiControl.bWriteParam
        toggle multiControl.bWriteParam
    ComboBoxTable (25,79 350x32), variable: multiControl.nMotorControlIndex, data array: multiControl.aMotorSelection
        p3854506369: multiControl.aMotorSelection[INDEX]
    Label (543,275 150x30), "MODE"
    Label (548,136 150x30), "INPUT"
    Label (543,412 150x30), "OUTPUT"
    Label (125,131 150x30), "STATUS"
    Rectangle (109,250 183x29), "DISABLED", colour toggle: multiControl.aStatusVar[3]
    Rectangle (109,219 183x29), "ERROR STOP", colour toggle: multiControl.aStatusVar[2]
    Rectangle (109,188 183x29), "ERROR ID:", colour toggle: multiControl.aMotorActive[1]
    Rectangle (109,157 183x29), "ERROR", colour toggle: multiControl.aStatusVar[1]
    Rectangle (108,343 183x29), "PROTECTED MODE", colour toggle: multiControl.aStatusVar[6]
    Rectangle (64,405 270x29), "MOTION COMMANDS LOCKED", colour toggle: multiControl.aStatusVar[8]
    Rectangle (74,436 250x29), "SOFT LIMIT MIN EXCEEDED", colour toggle: multiControl.aStatusVar[9]
    Rectangle (71,467 250x29), "SOFT LIMIT MAX EXCEEDED", colour toggle: multiControl.aStatusVar[10]
    Rectangle (71,498 250x29), "DRIVE DEVICE ERROR", colour toggle: multiControl.aStatusVar[11]
    Rectangle (109,529 183x29), "COUPLED", colour toggle: multiControl.aStatusVar[12]
    Button (418,70 392x54), "Variable Index: %3.0d", text variable: multiControl.nParameterIndex
        OnMouseClick: write the text variable via VisuDialogs.Numpad
END_VISUALIZATION

// ---- VISUs/VISUs/multiControlScreens/multiControlHelp.TcVIS
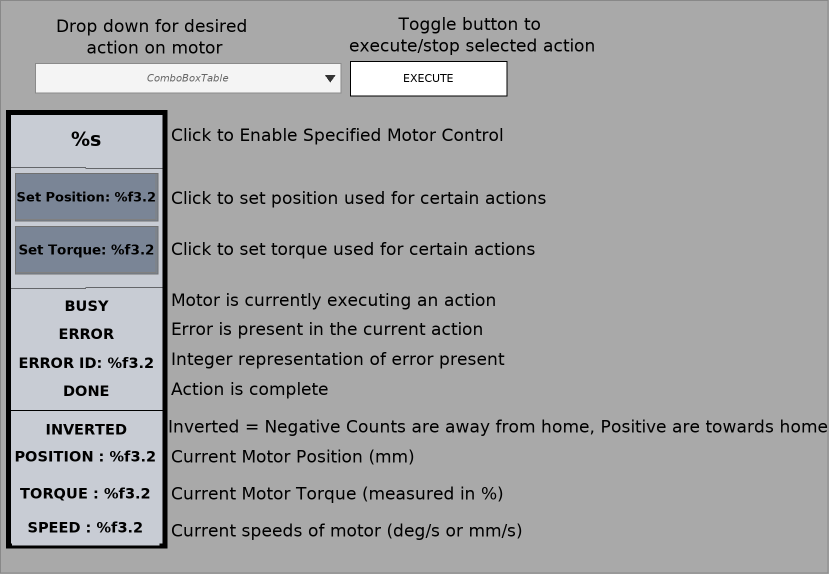
VISUALIZATION multiControlHelp  // 829x574
    Label (168,115 649x40), "Click to Enable Specified Motor Control"
    Label (168,178 649x40), "Click to set position used for certain actions"
    Label (168,229 649x40), "Click to set torque used for certain actions"
    Label (168,280 649x40), "Motor is currently executing an action"
    Label (168,309 649x40), "Error is present in the current action"
    Label (168,339 649x40), "Integer representation of error present"
    Label (168,369 649x40), "Action is complete"
    Label (168,439 649x35), "Current Motor Position (mm)"
    Label (168,476 649x35), "Current Motor Torque (measured in %)"
    Label (168,513 649x35), "Current speeds of motor (deg/s or mm/s)"
    RoundedRectangle (350,61 157x35), "EXECUTE"
    ComboBoxTable (35,63 306x30), data array: multiControl.aActionList
        p3854506369: multiControl.aActionList[INDEX]
    Rectangle (6,110 161x438)
    RoundedRectangle (14,116 145x47), "%s"
    Rectangle (12,439 147x35), "POSITION : %f3.2"
    Rectangle (15,293 143x26), "BUSY"
    Rectangle (15,378 143x26), "DONE"
    Rectangle (15,321 143x26), "ERROR"
    Rectangle (15,350 143x26), "ERROR ID: %f3.2"
    Rectangle (12,476 147x35), "TORQUE : %f3.2"
    Rectangle (12,510 147x35), "SPEED : %f3.2"
    Button (15,173 143x48), "Set Position: %f3.2"
    Button (15,226 143x48), "Set Torque: %f3.2"
    Line (6,167) (165,168)
    Line (6,288) (165,287)
    Line (6,410) (167,410)
    Label (39,16 231x42), "Drop down for desired action on motor"
    Label (350,11 245x48), "Toggle button to execute/stop selected action"
    Rectangle (15,413 143x33), "INVERTED"
    Label (165,409 663x35), "Inverted = Negative Counts are away from home, Positive are towards home."
END_VISUALIZATION

// ---- VISUs/VISUs/multiControlScreens/multiControlScreen.TcVIS
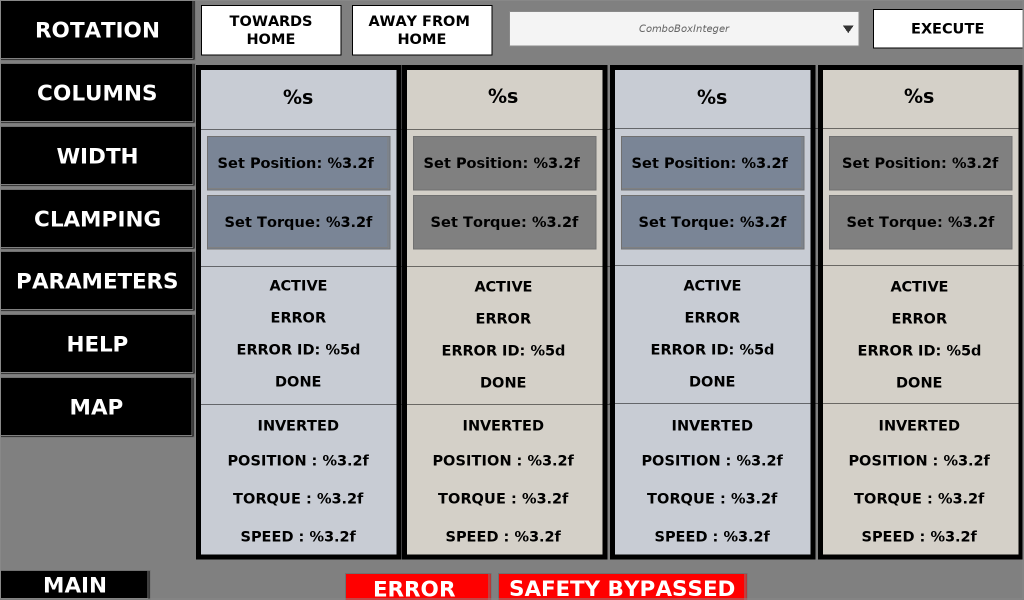
VISUALIZATION multiControlScreen  // 1024x600
    Button (0,570 150x30), "MAIN"
        OnMouseDown: change screen: mainScreen
        OnMouseDown: execute { GVL_machine.nPageIndex := 0; GVL_machine.bMotorsInitialized := FALSE; }
    Frame (196,0 829x574), frame switch variable: multiControl.multiCtrlFrameIndex
        shows motorControlScreen()
        shows machineMapScreen()
        shows multiControlHelp()
        shows parametersScreen()
        shows safetyResetScreen()
        shows tempEflexScreen()
        shows continueAutoScreen()
        shows rotationControl()
        shows widthControl()
    Button (0,0 195x60), "ROTATION", colour toggle: multiControl.nMotorControlIndex = 0
        toggle auto.bResetBtn
        OnMouseDown: execute { multiControl.multiCtrlFrameIndex :=0; multiControl.nMotorControlIndex := 0; }
    Button (498,573 249x31), "SAFETY BYPASSED", invisible if: NOT GVL_machine.bSafetyBypass
        OnMouseDown: change screen: safetyDisableWarning
    Button (345,573 146x32), "ERROR", invisible if: NOT GVL_machine.bDispErrorIcon
        OnMouseDown: change screen: errorScreen
    Button (0,63 195x60), "COLUMNS", colour toggle: multiControl.nMotorControlIndex = 2
        toggle auto.bResetBtn
        OnMouseDown: execute { multiControl.multiCtrlFrameIndex :=0; multiControl.nMotorControlIndex := 2; }
    Button (0,126 195x60), "WIDTH", colour toggle: multiControl.nMotorControlIndex = 3
        toggle auto.bResetBtn
        OnMouseDown: execute { multiControl.multiCtrlFrameIndex :=0; multiControl.nMotorControlIndex := 3; }
    Button (0,189 195x60), "CLAMPING", colour toggle: multiControl.nMotorControlIndex = 1
        toggle auto.bResetBtn
        OnMouseDown: execute { multiControl.multiCtrlFrameIndex :=0; multiControl.nMotorControlIndex := 1; }
    Button (0,314 195x60), "HELP", colour toggle: multiControl.multiCtrlFrameIndex = 2
        toggle auto.bResetBtn
        OnMouseDown: execute { multiControl.multiCtrlFrameIndex := 2; multiControl.nMotorControlIndex := 10; }
    Button (-1,377 195x60), "MAP", colour toggle: multiControl.multiCtrlFrameIndex = 1
        toggle auto.bResetBtn
        OnMouseDown: execute { multiControl.multiCtrlFrameIndex := 1; multiControl.nMotorControlIndex := 10; }
    Button (0,251 195x60), "PARAMETERS", colour toggle: multiControl.multiCtrlFrameIndex = 3
        toggle auto.bResetBtn
        OnMouseDown: execute { multiControl.multiCtrlFrameIndex :=3; multiControl.nMotorControlIndex := 10; }
END_VISUALIZATION

// ---- VISUs/VISUs/errorScreen.TcVIS
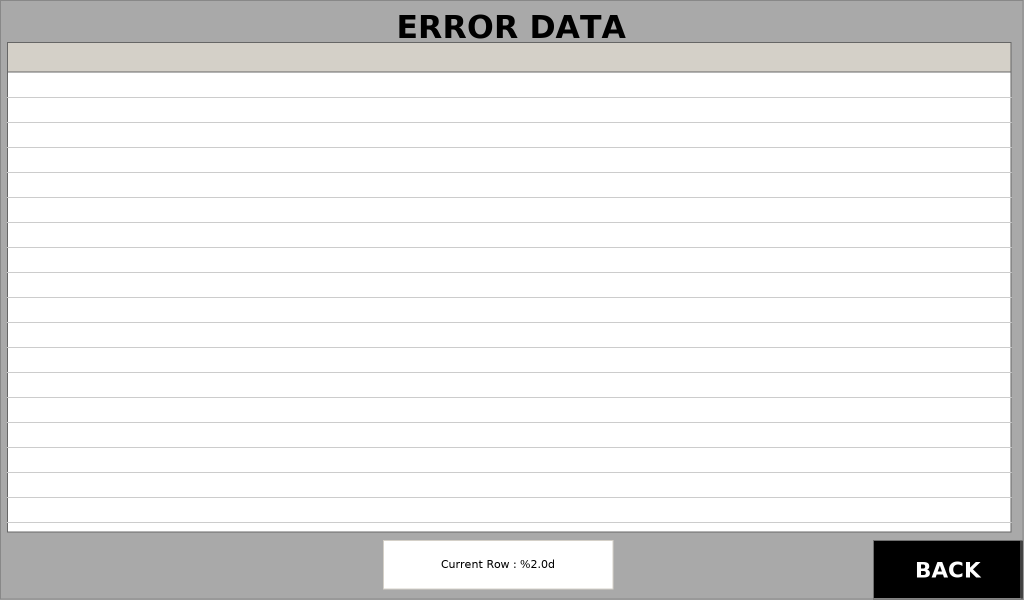
VISUALIZATION errorScreen  // 1024x600
    Label (0,10 1023x34), "ERROR DATA"
    Textfield (912,76 61x30)
    Textfield (834,76 61x30)
    Textfield (327,201 61x30)
    Textfield (555,75 84x30)
    Textfield (680,76 61x30)
    Table (7,42 1004x490), data array: GVL_machine.aErrorData
        p3854506369: GVL_machine.aErrorData[1,INDEX]
        p1892666644: GVL_machine.aErrorData[2,INDEX]
        p338671338: GVL_machine.aErrorData[3,INDEX]
        p1755163831: Function Block
        p2170511999: GVL_machine.aErrorData[4,INDEX]
        p3723444502: GVL_machine.aErrorData[5,INDEX]
        p2237128397: ERROR MESSAGE
    Button (873,540 150x60), "BACK"
        OnMouseDown: change screen: Previous maintenanceScreen3
        OnMouseDown: execute { GVL_machine.bDispErrorIcon := FALSE; }
    Textfield (383,540 230x49), "Current Row : %2.0d", text variable: GVL_machine.nErrorDataRow
END_VISUALIZATION

// ---- VISUs/VISUs/mainScreen.TcVIS
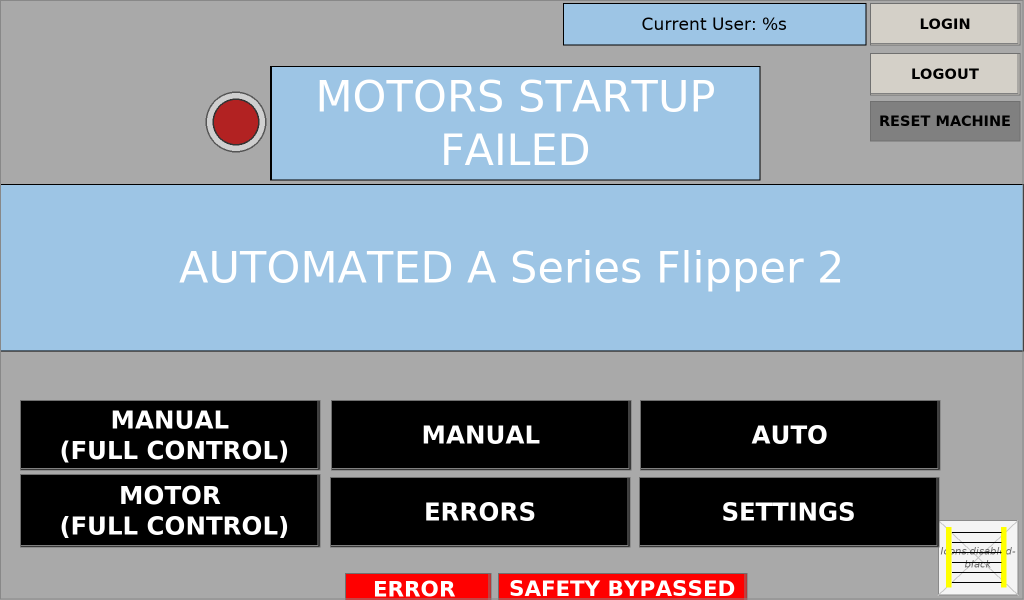
VISUALIZATION mainScreen  // 1024x600
    Image (938,520 80x75), invisible if: MAIN.bHideLtCurtainDisable, image: Icons.disabled-black
    Textfield (0,184 1024x167), "AUTOMATED A Series Flipper 2"
    Button (331,400 300x70), "MANUAL", invisible if: NOT GVL_machine.bMotorsInitialized
        OnMouseClick: change screen: manualScreen
        OnMouseClick: execute { GVL_machine.nPageIndex := 5; }
    Button (640,400 300x70), "AUTO", invisible if: NOT GVL_machine.bMotorsInitialized
        OnMouseClick: change screen: eflexScreen
        OnMouseClick: execute { GVL_machine.nPageIndex := 10; }
    Button (870,3 150x42), "LOGIN"
        OnMouseDown: VisuUserMgmt Type=Login
    Button (870,53 150x42), "LOGOUT"
        OnMouseDown: VisuUserMgmt Type=Logout
    Group (946,527 60x60), invisible if: GVL_machine.bSafetyBypass
        toggle GVL_machine.bMuteSafety
        Rectangle (0,0 5x60)
        Rectangle (55,0 5x60)
        Line (6,5) (55,5)
        Line (6,15) (55,15)
        Line (6,25) (55,25)
        Line (6,35) (55,35)
        Line (6,45) (55,45)
        Line (6,55) (55,55)
    Lamp1 (201,87 70x70), variable: NOT GVL_machine.bMotorsInitialized, invisible if: GVL_machine.bMotorsInitialized, style: Lamp-Lamp1-Red
    Textfield (270,66 489x114), "MOTORS STARTUP Please wait...", invisible if: GVL_machine.bMotorsInitialized
    Textfield (271,66 489x114), "MOTORS STARTUP FAILED", invisible if: NOT GVL_machine.bMotorInitFailedDisp
    Button (498,573 249x31), "SAFETY BYPASSED", invisible if: NOT GVL_machine.bSafetyBypass
        OnMouseDown: change screen: safetyDisableWarning
    Button (330,477 300x70), "ERRORS", invisible if: NOT GVL_machine.bMotorsInitialized
        OnMouseClick: change screen: errorScreen
    Button (639,477 300x70), "SETTINGS", invisible if: NOT GVL_machine.bMotorsInitialized
        OnMouseClick: change screen: settingsScreen
    Button (345,573 146x32), "ERROR", invisible if: NOT GVL_machine.bDispErrorIcon
        OnMouseDown: change screen: errorScreen
    Button (20,400 300x70), "MANUAL (FULL CONTROL)", invisible if: NOT GVL_machine.bMotorsInitialized
        OnMouseClick: change screen: manualBypassedScreen
        OnMouseClick: execute { GVL_machine.nPageIndex := 5; }
    Textfield (563,3 303x42), "Current User: %s", text variable: VisuElems.CurrentUserName
    Button (870,101 150x40), "RESET MACHINE"
        OnMouseDown: toggle GVL_machine.bResetMachine
    Button (20,474 300x73), "MOTOR (FULL CONTROL)", invisible if: NOT GVL_machine.bMotorsInitialized
        OnMouseClick: change screen: multiControlScreen
        OnMouseClick: execute { GVL_machine.nPageIndex := 20; }
END_VISUALIZATION

// ---- VISUs/VISUs/multiControlScreens/machineMapScreen.TcVIS
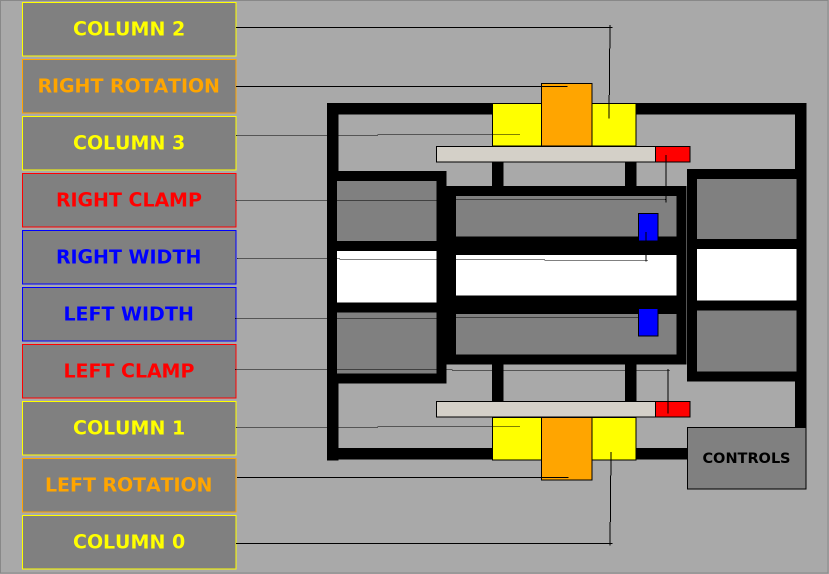
VISUALIZATION machineMapScreen  // 829x574
    Group (327,83 479x406)
        Rectangle (165,20 11x357)
        Rectangle (298,20 11x357)
        Rectangle (119,103 240x60)
        Rectangle (119,221 240x60)
        Rectangle (1,20 478x11)
        Rectangle (0,365 478x11)
        Rectangle (0,20 11x357)
        Rectangle (468,20 11x357)
        Rectangle (0,88 119x89)
        Rectangle (0,211 119x89)
        Rectangle (0,158 119x71)
        Rectangle (360,86 119x89)
        Rectangle (360,209 119x89)
        Rectangle (360,156 119x71)
        Rectangle (119,162 240x60)
        Rectangle (360,344 119x62), "CONTROLS"
        Rectangle (165,20 51x43)
        Rectangle (258,20 51x43)
        Rectangle (214,0 51x63)
        Rectangle (109,63 231x16)
        Rectangle (328,63 35x16)
        Rectangle (165,334 51x43)
        Rectangle (258,334 51x43)
        Rectangle (214,334 51x63)
        Rectangle (109,318 231x16)
        Rectangle (328,318 35x16)
    Rectangle (22,2 214x54), "COLUMN 2"
    Rectangle (22,59 214x54), "RIGHT ROTATION"
    Rectangle (22,116 214x54), "COLUMN 3"
    Rectangle (22,173 214x54), "RIGHT CLAMP"
    Rectangle (22,230 214x54), "RIGHT WIDTH"
    Rectangle (22,287 214x54), "LEFT WIDTH"
    Rectangle (22,344 214x54), "LEFT CLAMP"
    Rectangle (22,401 214x54), "COLUMN 1"
    Rectangle (22,515 214x54), "COLUMN 0"
    Rectangle (22,458 214x54), "LEFT ROTATION"
    Line (236,27) (612,27)
    Line (609,118) (610,25)
    Line (236,86) (567,86)
    Line (236,135) (519,134)
    Line (236,200) (665,199)
    Line (237,258) (647,260)
    Line (235,318) (640,317)
    Line (235,369) (669,370)
    Rectangle (638,213 20x28)
    Rectangle (638,308 20x28)
    Line (666,202) (666,155)
    Line (646,261) (646,232)
    Line (668,413) (668,369)
    Line (236,427) (519,426)
    Line (236,543) (612,543)
    Line (610,545) (611,452)
    Line (237,477) (568,477)
END_VISUALIZATION

// ---- VISUs/VISUs/multiControlScreens/motorControlScreen.TcVIS
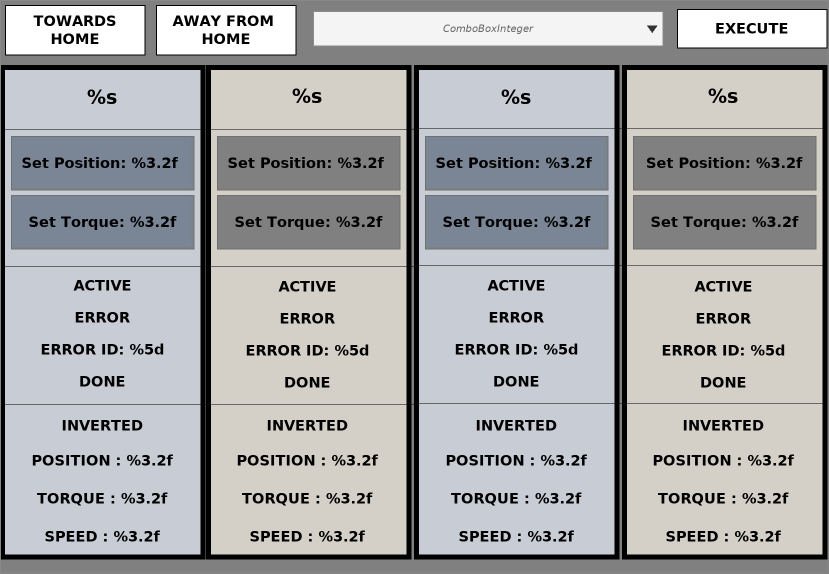
VISUALIZATION motorControlScreen  // 829x574
    Rectangle (206,65 205x494)
    RoundedRectangle (677,9 150x39), "EXECUTE", colour toggle: multiControl.bExecute
        toggle multiControl.bExecute
    Rectangle (0,65 205x494)
    Rectangle (414,65 205x494)
    Rectangle (622,65 205x494)
    RoundedRectangle (10,71 185x53), "%s", text variable: multiControl.sMotorDisp1, colour toggle: multiControl.aMotorEnable[1]
        p55702900: multiControl.aDispFontColor[1]
        toggle multiControl.aMotorEnable[1]
    Rectangle (11,443 183x35), "POSITION : %3.2f", text variable: multiControl.aMotorPos[1]
    Rectangle (11,271 183x29), "ACTIVE", colour toggle: multiControl.aMotorActive[1]
    Rectangle (11,367 183x29), "DONE", colour toggle: multiControl.aMotorDone[1]
    Rectangle (11,303 183x29), "ERROR", colour toggle: multiControl.aMotorError[1]
    Rectangle (11,335 183x29), "ERROR ID: %5d", text variable: multiControl.aMotorErrorId[1]
    Rectangle (11,481 183x35), "TORQUE : %3.2f", text variable: multiControl.aMotorTorque[1]
    Rectangle (11,519 183x35), "SPEED : %3.2f", text variable: multiControl.aMotorSpeed[1]
    Button (11,136 183x54), "Set Position: %3.2f", text variable: multiControl.aMotorSetPos[1], invisible if: multiControl.bHideSetPos
        OnMouseClick: write the text variable via VisuDialogs.Numpad
    Button (11,195 183x54), "Set Torque: %3.2f", text variable: multiControl.aMotorSetTorq[1], invisible if: multiControl.bHideSetTorq
        OnMouseClick: write the text variable via VisuDialogs.Numpad
    Line (0,129) (827,128)
    Line (1,266) (828,265)
    Line (0,404) (827,403)
    Button (217,195 183x54), "Set Torque: %3.2f", text variable: multiControl.aMotorSetTorq[2], invisible if: multiControl.bHideSetTorq
        OnMouseClick: write the text variable via VisuDialogs.Numpad
    Button (217,136 183x54), "Set Position: %3.2f", text variable: multiControl.aMotorSetPos[2], invisible if: multiControl.bHideSetPos
        OnMouseClick: write the text variable via VisuDialogs.Numpad
    RoundedRectangle (215,70 185x53), "%s", text variable: multiControl.sMotorDisp2, colour toggle: multiControl.aMotorEnable[2]
        p55702900: multiControl.aDispFontColor[2]
        toggle multiControl.aMotorEnable[2]
    Rectangle (216,272 183x29), "ACTIVE", colour toggle: multiControl.aMotorActive[2]
    Rectangle (216,443 183x35), "POSITION : %3.2f", text variable: multiControl.aMotorPos[2]
    Rectangle (216,368 183x29), "DONE", colour toggle: multiControl.aMotorDone[2]
    Rectangle (216,304 183x29), "ERROR", colour toggle: multiControl.aMotorError[2]
    Rectangle (216,336 183x29), "ERROR ID: %5d", text variable: multiControl.aMotorErrorId[2]
    Rectangle (216,481 183x35), "TORQUE : %3.2f", text variable: multiControl.aMotorTorque[2]
    Rectangle (216,519 183x35), "SPEED : %3.2f", text variable: multiControl.aMotorSpeed[2]
    RoundedRectangle (424,71 185x53), "%s", text variable: multiControl.sMotorDisp3, colour toggle: multiControl.aMotorEnable[3], invisible if: multiControl.bHideDispMotor3
        p55702900: multiControl.aDispFontColor[3]
        toggle multiControl.aMotorEnable[3]
    Rectangle (425,443 183x35), "POSITION : %3.2f", text variable: multiControl.aMotorPos[3], invisible if: multiControl.bHideDispMotor3
    Rectangle (425,271 183x29), "ACTIVE", colour toggle: multiControl.aMotorActive[3], invisible if: multiControl.bHideDispMotor3
    Rectangle (425,367 183x29), "DONE", colour toggle: multiControl.aMotorDone[3], invisible if: multiControl.bHideDispMotor3
    Rectangle (425,303 183x29), "ERROR", colour toggle: multiControl.aMotorError[3], invisible if: multiControl.bHideDispMotor3
    Rectangle (425,335 183x29), "ERROR ID: %5d", text variable: multiControl.aMotorErrorId[3], invisible if: multiControl.bHideDispMotor3
    Rectangle (425,481 183x35), "TORQUE : %3.2f", text variable: multiControl.aMotorTorque[3], invisible if: multiControl.bHideDispMotor3
    Rectangle (425,519 183x35), "SPEED : %3.2f", text variable: multiControl.aMotorSpeed[3], invisible if: multiControl.bHideDispMotor3
    Button (425,136 183x54), "Set Position: %3.2f", text variable: multiControl.aMotorSetPos[3], invisible if: multiControl.bHideDispMotor3 OR multiControl.bHideSetPos
        OnMouseClick: write the text variable via VisuDialogs.Numpad
    Button (425,195 183x54), "Set Torque: %3.2f", text variable: multiControl.aMotorSetTorq[3], invisible if: multiControl.bHideDispMotor3 OR multiControl.bHideSetTorq
        OnMouseClick: write the text variable via VisuDialogs.Numpad
    RoundedRectangle (631,70 185x53), "%s", text variable: multiControl.sMotorDisp4, colour toggle: multiControl.aMotorEnable[4], invisible if: multiControl.bHideDispMotor4
        p55702900: multiControl.aDispFontColor[4]
        toggle multiControl.aMotorEnable[4]
    Button (633,195 183x54), "Set Torque: %3.2f", text variable: multiControl.aMotorSetTorq[4], invisible if: multiControl.bHideDispMotor4 OR multiControl.bHideSetTorq
        OnMouseClick: write the text variable via VisuDialogs.Numpad
    Button (633,136 183x54), "Set Position: %3.2f", text variable: multiControl.aMotorSetPos[4], invisible if: multiControl.bHideDispMotor4 OR multiControl.bHideSetPos
        OnMouseClick: write the text variable via VisuDialogs.Numpad
    Rectangle (632,272 183x29), "ACTIVE", colour toggle: multiControl.aMotorActive[4], invisible if: multiControl.bHideDispMotor4
    Rectangle (632,443 183x35), "POSITION : %3.2f", text variable: multiControl.aMotorPos[4], invisible if: multiControl.bHideDispMotor4
    Rectangle (632,368 183x29), "DONE", colour toggle: multiControl.aMotorDone[4], invisible if: multiControl.bHideDispMotor4
    Rectangle (632,304 183x29), "ERROR", colour toggle: multiControl.aMotorError[4], invisible if: multiControl.bHideDispMotor4
    Rectangle (632,336 183x29), "ERROR ID: %5d", text variable: multiControl.aMotorErrorId[4], invisible if: multiControl.bHideDispMotor4
    Rectangle (632,481 183x35), "TORQUE : %3.2f", text variable: multiControl.aMotorTorque[4], invisible if: multiControl.bHideDispMotor4
    Rectangle (632,519 183x35), "SPEED : %3.2f", text variable: multiControl.aMotorSpeed[4], invisible if: multiControl.bHideDispMotor4
    RoundedRectangle (5,5 140x50), "TOWARDS HOME", colour toggle: multiControl.bHomeDirection, invisible if: multiControl.bHideDirection
        toggle multiControl.bHomeDirection
    RoundedRectangle (156,5 140x50), "AWAY FROM HOME", colour toggle: NOT multiControl.bHomeDirection, invisible if: multiControl.bHideDirection
        toggle multiControl.bHomeDirection
    Rectangle (11,411 183x29), "INVERTED", colour toggle: multiControl.aMotorInverted[1]
    Rectangle (425,411 183x29), "INVERTED", colour toggle: multiControl.aMotorInverted[3], invisible if: multiControl.bHideDispMotor3
    Rectangle (216,411 183x29), "INVERTED", colour toggle: multiControl.aMotorInverted[2]
    Rectangle (632,411 183x29), "INVERTED", colour toggle: multiControl.aMotorInverted[4], invisible if: multiControl.bHideDispMotor4
    ComboBoxInteger (313,11 350x35), variable: multiControl.nActionIndex, text list: 'actionSelectList'
END_VISUALIZATION

// ---- VISUs/VISUs/manualBypassedScreen.TcVIS
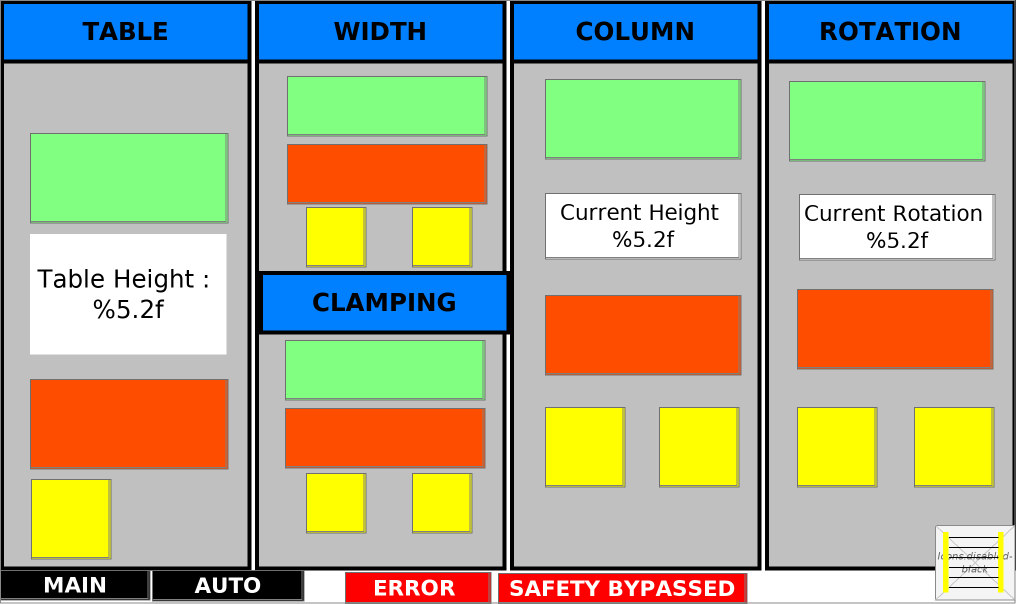
VISUALIZATION manualBypassedScreen  // 1016x604
    Group (0,0 1016x570)
        Rectangle (255,0 251x570)
        Rectangle (510,0 251x570)
        Rectangle (765,0 251x570)
        Rectangle (0,0 251x570)
    Button (545,79 196x80), image: Icons.up-black
        OnMouseDown: execute { manual.eColumnState := 1; }
        OnMouseUp: execute { manual.eColumnState := 0; }
    Button (545,295 196x80), image: Icons.down-black
        OnMouseDown: execute { manual.eColumnState := 2; }
        OnMouseUp: execute { manual.eColumnState := 0; }
    Button (797,289 196x80), image: Icons.rotate-ccw-black
        OnMouseDown: execute { manual.eRotationState := 1; }
        OnMouseUp: execute { manual.eRotationState := 0; }
    Button (789,81 196x80), image: Icons.rotate-cw-black
        OnMouseDown: execute { manual.eRotationState := 2; }
        OnMouseUp: execute { manual.eRotationState := 0; }
    Button (545,407 80x80), image: Icons.home-black
        OnMouseDown: execute { manual.eColumnState := 4; }
    Button (797,407 80x80), image: Icons.home-black
        OnMouseDown: execute { manual.eRotationState := 4; }
    Button (659,407 80x80), image: Icons.reset-black
        OnMouseDown: execute { manual.eColumnState := 3; }
    Button (914,407 80x80), image: Icons.reset-black
        OnMouseDown: execute { manual.eRotationState := 3; }
    Button (412,473 60x60), image: Icons.reset-black
        OnMouseDown: execute { manual.eClampingState := 3; }
    Button (287,76 200x60), image: Icons.width-in-black
        OnMouseDown: execute { manual.eWidthState := 1; }
        OnMouseUp: execute { manual.eWidthState := 0; }
    Button (287,144 200x60), image: Icons.width-out-black
        OnMouseDown: execute { manual.eWidthState := 2; }
        OnMouseUp: execute { manual.eWidthState := 0; }
    Button (285,340 200x60), image: Icons.Unclamp-black
        OnMouseDown: execute { manual.eClampingState := 1; }
        OnMouseUp: execute { manual.eClampingState := 0; }
    Button (285,408 200x60), image: Icons.clamp-black
        OnMouseDown: execute { manual.eClampingState := 2; }
        OnMouseUp: execute { manual.eClampingState := 0; }
    Button (306,473 60x60), image: Icons.home-black
        OnMouseDown: execute { manual.eClampingState := 4; }
    Button (306,207 60x60), image: Icons.home-black
        OnMouseDown: execute { manual.eWidthState := 4; }
    Button (412,207 60x60), image: Icons.reset-black
        OnMouseDown: execute { manual.eWidthState := 3; }
    Button (30,379 198x90), image: Icons.down-black
        OnMouseDown: execute { manual.eTableState := 2; }
        OnMouseUp: execute { manual.eTableState := 0; }
    RoundedRectangle (0,0 251x63), "TABLE", colour toggle: manual.bTableMoveStatus
    RoundedRectangle (255,0 251x63), "WIDTH", colour toggle: manual.bWidthMoveStatus
    RoundedRectangle (510,0 251x63), "COLUMN", colour toggle: manual.bColumnMoveStatus
    RoundedRectangle (765,0 251x63), "ROTATION", colour toggle: manual.bRotationMoveStatus
    Button (30,133 198x90), image: Icons.up-black
        OnMouseDown: execute { manual.eTableState := 1; }
        OnMouseUp: execute { manual.eTableState := 0; }
    RoundedRectangle (30,234 196x120), "Table Height : %5.2f", text variable: GVL_ignition.fTableHeight
    Button (545,193 196x66), "Current Height %5.2f", text variable: GVL_ignition.fColumnHeight
    RoundedRectangle (259,271 251x63), "CLAMPING", colour toggle: manual.bClampingMoveStatus
    Button (0,570 150x30), "MAIN"
        OnMouseDown: change screen: mainScreen
        OnMouseDown: execute { GVL_machine.nPageIndex := 0; }
    Button (152,570 152x31), "AUTO"
        OnMouseDown: change screen: eflexScreen
        OnMouseDown: execute { GVL_machine.nPageIndex := 10; }
    Button (799,194 196x66), "Current Rotation %5.2f", text variable: GVL_ignition.fRotationDistance
    Button (31,479 80x80), image: Icons.home-black
        OnMouseDown: execute { manual.eTableState := 4; }
    Image (935,525 80x75), invisible if: MAIN.bHideLtCurtainDisable, image: Icons.disabled-black
    Group (943,532 60x60), invisible if: GVL_machine.bSafetyBypass
        toggle GVL_machine.bMuteSafety
        Rectangle (0,0 5x60)
        Rectangle (55,0 5x60)
        Line (6,5) (55,5)
        Line (6,15) (55,15)
        Line (6,25) (55,25)
        Line (6,35) (55,35)
        Line (6,45) (55,45)
        Line (6,55) (55,55)
    Button (498,573 249x31), "SAFETY BYPASSED", invisible if: NOT GVL_machine.bSafetyBypass
        OnMouseDown: change screen: safetyDisableWarning
    Button (345,572 146x32), "ERROR", invisible if: NOT GVL_machine.bDispErrorIcon
        OnMouseDown: change screen: errorScreen
END_VISUALIZATION

// ---- VISUs/VISUs/manualScreen.TcVIS
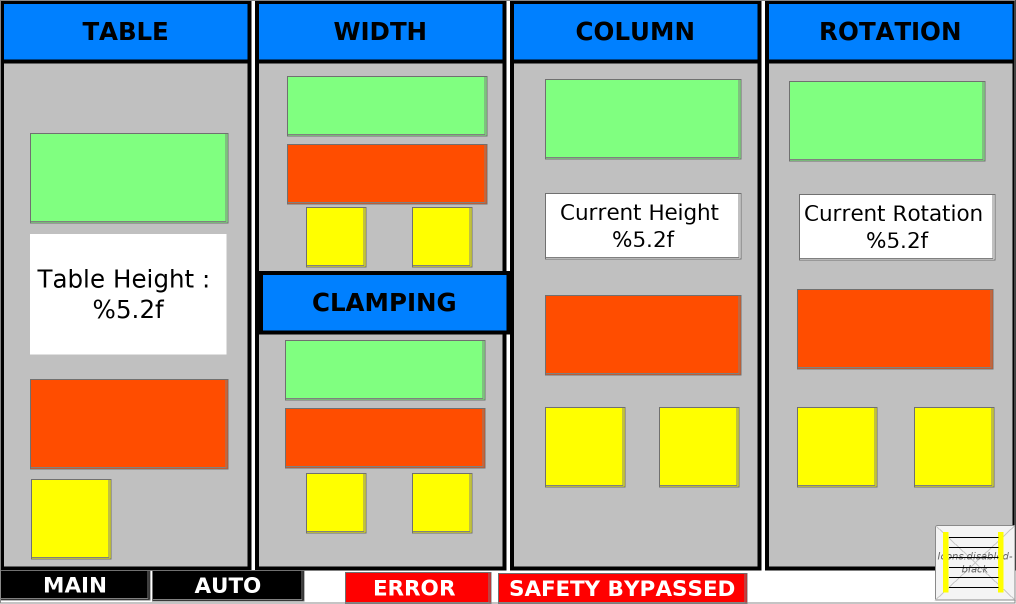
VISUALIZATION manualScreen  // 1016x604
    Group (0,0 1016x570)
        Rectangle (255,0 251x570)
        Rectangle (510,0 251x570)
        Rectangle (765,0 251x570)
        Rectangle (0,0 251x570)
    Button (545,79 196x80), invisible if: manual.bHideColumnBtns, image: Icons.up-black
        OnMouseDown: execute { manual.eColumnState := 1; }
        OnMouseUp: execute { manual.eColumnState := 0; }
    Button (545,295 196x80), invisible if: manual.bHideColumnBtns, image: Icons.down-black
        OnMouseDown: execute { manual.eColumnState := 2; }
        OnMouseUp: execute { manual.eColumnState := 0; }
    Button (797,289 196x80), invisible if: manual.bHideRotationBtns, image: Icons.rotate-ccw-black
        OnMouseDown: execute { manual.eRotationState := 1; }
        OnMouseUp: execute { manual.eRotationState := 0; }
    Button (789,81 196x80), invisible if: manual.bHideRotationBtns, image: Icons.rotate-cw-black
        OnMouseDown: execute { manual.eRotationState := 2; }
        OnMouseUp: execute { manual.eRotationState := 0; }
    Button (545,407 80x80), image: Icons.home-black
        OnMouseDown: execute { manual.eColumnState := 4; }
    Button (797,407 80x80), image: Icons.home-black
        OnMouseDown: execute { manual.eRotationState := 4; }
    Button (659,407 80x80), image: Icons.reset-black
        OnMouseDown: execute { manual.eColumnState := 3; }
    Button (914,407 80x80), image: Icons.reset-black
        OnMouseDown: execute { manual.eRotationState := 3; }
    Button (412,473 60x60), image: Icons.reset-black
        OnMouseDown: execute { manual.eClampingState := 3; }
    Button (287,76 200x60), invisible if: manual.bHideWidthBtns, image: Icons.width-in-black
        OnMouseDown: execute { manual.eWidthState := 1; }
        OnMouseUp: execute { manual.eWidthState := 0; }
    Button (287,144 200x60), invisible if: manual.bHideWidthBtns, image: Icons.width-out-black
        OnMouseDown: execute { manual.eWidthState := 2; }
        OnMouseUp: execute { manual.eWidthState := 0; }
    Button (285,340 200x60), invisible if: manual.bHideClampingBtns, image: Icons.Unclamp-black
        OnMouseDown: execute { manual.eClampingState := 1; }
        OnMouseUp: execute { manual.eClampingState := 0; }
    Button (285,408 200x60), invisible if: manual.bHideClampingBtns, image: Icons.clamp-black
        OnMouseDown: execute { manual.eClampingState := 2; }
        OnMouseUp: execute { manual.eClampingState := 0; }
    Button (306,473 60x60), image: Icons.home-black
        OnMouseDown: execute { manual.eClampingState := 4; }
    Button (306,207 60x60), image: Icons.home-black
        OnMouseDown: execute { manual.eWidthState := 4; }
    Button (412,207 60x60), image: Icons.reset-black
        OnMouseDown: execute { manual.eWidthState := 3; }
    Button (30,379 198x90), invisible if: manual.bHideTableBtns, image: Icons.down-black
        OnMouseDown: execute { manual.eTableState := 2; }
        OnMouseUp: execute { manual.eTableState := 0; }
    RoundedRectangle (0,0 251x63), "TABLE", colour toggle: manual.bTableMoveStatus
    RoundedRectangle (255,0 251x63), "WIDTH", colour toggle: manual.bWidthMoveStatus
    RoundedRectangle (510,0 251x63), "COLUMN", colour toggle: manual.bColumnMoveStatus
    RoundedRectangle (765,0 251x63), "ROTATION", colour toggle: manual.bRotationMoveStatus
    Button (30,133 198x90), invisible if: manual.bHideTableBtns, image: Icons.up-black
        OnMouseDown: execute { manual.eTableState := 1; }
        OnMouseUp: execute { manual.eTableState := 0; }
    RoundedRectangle (30,234 196x120), "Table Height : %5.2f", text variable: GVL_ignition.fTableHeight
    Button (545,193 196x66), "Current Height %5.2f", text variable: GVL_ignition.fColumnHeight
    RoundedRectangle (259,271 251x63), "CLAMPING", colour toggle: manual.bClampingMoveStatus
    Button (0,570 150x30), "MAIN"
        OnMouseDown: change screen: mainScreen
        OnMouseDown: execute { GVL_machine.nPageIndex := 0; }
    Button (152,570 152x31), "AUTO"
        OnMouseDown: change screen: eflexScreen
        OnMouseDown: execute { GVL_machine.nPageIndex := 10; }
    Button (799,194 196x66), "Current Rotation %5.2f", text variable: GVL_ignition.fRotationDistance
    Button (31,479 80x80), image: Icons.home-black
        OnMouseDown: execute { manual.eTableState := 4; }
    Image (935,525 80x75), invisible if: MAIN.bHideLtCurtainDisable, image: Icons.disabled-black
    Group (943,532 60x60), invisible if: GVL_machine.bSafetyBypass
        toggle GVL_machine.bMuteSafety
        Rectangle (0,0 5x60)
        Rectangle (55,0 5x60)
        Line (6,5) (55,5)
        Line (6,15) (55,15)
        Line (6,25) (55,25)
        Line (6,35) (55,35)
        Line (6,45) (55,45)
        Line (6,55) (55,55)
    Button (498,573 249x31), "SAFETY BYPASSED", invisible if: NOT GVL_machine.bSafetyBypass
        OnMouseDown: change screen: safetyDisableWarning
    Button (345,572 146x32), "ERROR", invisible if: NOT GVL_machine.bDispErrorIcon
        OnMouseDown: change screen: errorScreen
END_VISUALIZATION

// ---- VISUs/VISUs/safetyDisableWarning.TcVIS
